LIN {X 0,Y 404.496,Z 624.581,A -85,B 0,C 180,E1 -11091.801,E2 -11091.801} C_VEL
LIN {X 0,Y 405.836,Z 611.424,A -85,B 0,C 180,E1 -11092.797,E2 -11092.797} C_VEL
LIN {X 0,Y 407.026,Z 596.699,A -85,B 0,C 180,E1 -11093.683,E2 -11093.683} C_VEL
LIN {X 0,Y 408.001,Z 581.797,A -85,B 0,C 180,E1 -11094.357,E2 -11094.357} C_VEL
LIN {X 0,Y 408.768,Z 566.165,A -85,B 0,C 180,E1 -11094.844,E2 -11094.844} C_VEL
LIN {X 0,Y 409.775,Z 521.843,A -85,B 0,C 180,E1 -11095.662,E2 -11095.662} C_VEL
LIN {X 0,Y 411.509,Z 429.898,A -85,B 0,C 180,E1 -11097.306,E2 -11097.306} C_VEL
LIN {X 0,Y 405.614,Z 399.49,A -85,B 0,C 180,E1 -11098.332,E2 -11098.332} C_VEL
LIN {X 0,Y 405.096,Z 396.543,A -85,B 0,C 180,E1 -11098.473,E2 -11098.473} C_VEL
LIN {X 0,Y 405.534,Z 388.379,A -85,B 0,C 180,E1 -11099.611,E2 -11099.611} C_VEL
LIN {X 0,Y 402.994,Z 376.938,A -85,B 0,C 180,E1 -11101.546,E2 -11101.546} C_VEL
LIN {X 0,Y 398.838,Z 361.587,A -85,B 0,C 180,E1 -11104.324,E2 -11104.324} C_VEL
LIN {X 0,Y 397.121,Z 355.796,A -85,B 0,C 180,E1 -11105.447,E2 -11105.447} C_VEL
LIN {X 0,Y 397.087,Z 355.636,A -85,B 0,C 180,E1 -11108.853,E2 -11108.853} C_VEL
LIN {X 0,Y 397.053,Z 355.648,A -85,B 0,C 180,E1 -11112.269,E2 -11112.269} C_VEL
LIN {X 0,Y 397.084,Z 355.643,A -85,B 0,C 180,E1 -11115.069,E2 -11115.069} C_VEL
LIN {X 0,Y 397.051,Z 355.65,A -85,B 0,C 180,E1 -11118.024,E2 -11118.024} C_VEL
LIN {X 0,Y 397.089,Z 355.644,A -85,B 0,C 180,E1 -11121.723,E2 -11121.723} C_VEL
LIN {X 0,Y 397.119,Z 355.639,A -85,B 0,C 180,E1 -11125.506,E2 -11125.506} C_VEL
LIN {X 0,Y 397.077,Z 355.639,A -85,B 0,C 180,E1 -11129.117,E2 -11129.117} C_VEL
LIN {X 0,Y 397.099,Z 355.633,A -85,B 0,C 180,E1 -11132.603,E2 -11132.603} C_VEL
LIN {X 0,Y 397.112,Z 355.641,A -85,B 0,C 180,E1 -11135.98,E2 -11135.98} C_VEL
LIN {X 0,Y 397.139,Z 355.64,A -85,B 0,C 180,E1 -11139.705,E2 -11139.705} C_VEL
LIN {X 0,Y 397.182,Z 355.622,A -85,B 0,C 180,E1 -11142.845,E2 -11142.845} C_VEL
LIN {X 0,Y 397.229,Z 355.627,A -85,B 0,C 180,E1 -11146.703,E2 -11146.703} C_VEL
LIN {X 0,Y 397.216,Z 355.619,A -85,B 0,C 180,E1 -11149.809,E2 -11149.809} C_VEL
LIN {X 0,Y 397.335,Z 355.615,A -85,B 0,C 180,E1 -11152.888,E2 -11152.888} C_VEL
LIN {X 0,Y 397.248,Z 355.611,A -85,B 0,C 180,E1 -11154.925,E2 -11154.925} C_VEL
LIN {X 0,Y 397.446,Z 355.602,A -85,B 0,C 180,E1 -11157.973,E2 -11157.973} C_VEL
LIN {X 0,Y 397.577,Z 355.577,A -85,B 0,C 180,E1 -11160,E2 -11160} C_VEL
LIN {X 0,Y 397.37,Z 355.602,A -85,B 0,C 180,E1 -11163.041,E2 -11163.041} C_VEL
LIN {X 0,Y 397.346,Z 355.607,A -85,B 0,C 180,E1 -11166.092,E2 -11166.092} C_VEL
LIN {X 0,Y 397.236,Z 355.617,A -85,B 0,C 180,E1 -11169.162,E2 -11169.162} C_VEL
LIN {X 0,Y 397.22,Z 355.622,A -85,B 0,C 180,E1 -11172.258,E2 -11172.258} C_VEL
LIN {X 0,Y 397.179,Z 355.629,A -85,B 0,C 180,E1 -11175.392,E2 -11175.392} C_VEL
LIN {X 0,Y 397.158,Z 355.631,A -85,B 0,C 180,E1 -11178.574,E2 -11178.574} C_VEL
LIN {X 0,Y 397.109,Z 355.644,A -85,B 0,C 180,E1 -11181.818,E2 -11181.818} C_VEL
LIN {X 0,Y 397.152,Z 355.629,A -85,B 0,C 180,E1 -11185.512,E2 -11185.512} C_VEL
LIN {X 0,Y 397.123,Z 355.642,A -85,B 0,C 180,E1 -11188.543,E2 -11188.543} C_VEL
LIN {X 0,Y 397.078,Z 355.647,A -85,B 0,C 180,E1 -11192.071,E2 -11192.071} C_VEL
LIN {X 0,Y 397.119,Z 355.642,A -85,B 0,C 180,E1 -11195.503,E2 -11195.503} C_VEL
LIN {X 0,Y 397.126,Z 355.616,A -85,B 0,C 180,E1 -11198.861,E2 -11198.861} C_VEL
LIN {X 0,Y 397.071,Z 355.64,A -85,B 0,C 180,E1 -11202.267,E2 -11202.267} C_VEL
LIN {X 0,Y 397.088,Z 355.635,A -85,B 0,C 180,E1 -11205.068,E2 -11205.068} C_VEL
LIN {X 0,Y 397.065,Z 355.633,A -85,B 0,C 180,E1 -11208.021,E2 -11208.021} C_VEL
LIN {X 0,Y 397.131,Z 355.645,A -85,B 0,C 180,E1 -11211.138,E2 -11211.138} C_VEL
LIN {X 0,Y 397.154,Z 355.714,A -85,B 0,C 180,E1 -11215.124,E2 -11215.124} C_VEL
LIN {X 0,Y 397.314,Z 356.566,A -85,B 0,C 180,E1 -11215.372,E2 -11215.372} C_VEL
LIN {X 0,Y 401.916,Z 373.552,A -85,B 0,C 180,E1 -11218.529,E2 -11218.529} C_VEL
LIN {X 0,Y 405.39,Z 387.316,A -85,B 0,C 180,E1 -11220.96,E2 -11220.96} C_VEL
LIN {X 0,Y 405.046,Z 393.159,A -85,B 0,C 180,E1 -11221.805,E2 -11221.805} C_VEL
LIN {X 0,Y 410.902,Z 428.294,A -85,B 0,C 180,E1 -11222.931,E2 -11222.931} C_VEL
LIN {X 0,Y 408.199,Z 565.443,A -85,B 0,C 180,E1 -11225.39,E2 -11225.39} C_VEL
LIN {X 0,Y 407.442,Z 581.285,A -85,B 0,C 180,E1 -11225.88,E2 -11225.88} C_VEL
LIN {X 0,Y 406.442,Z 596.437,A -85,B 0,C 180,E1 -11226.565,E2 -11226.565} C_VEL
LIN {X 0,Y 405.3,Z 610.9,A -85,B 0,C 180,E1 -11227.44,E2 -11227.44} C_VEL
LIN {X 0,Y 403.993,Z 624.081,A -85,B 0,C 180,E1 -11228.439,E2 -11228.439} C_VEL
LIN {X 0,Y 402.589,Z 637.469,A -85,B 0,C 180,E1 -11229.699,E2 -11229.699} C_VEL
LIN {X 0,Y 401.232,Z 649.387,A -85,B 0,C 180,E1 -11231.061,E2 -11231.061} C_VEL
LIN {X 0,Y 399.9,Z 660.685,A -85,B 0,C 180,E1 -11232.617,E2 -11232.617} C_VEL
LIN {X 0,Y 398.64,Z 671.405,A -85,B 0,C 180,E1 -11234.404,E2 -11234.404} C_VEL
LIN {X 0,Y 397.674,Z 680.308,A -85,B 0,C 180,E1 -11236.198,E2 -11236.198} C_VEL
LIN {X 0,Y 396.924,Z 688.618,A -85,B 0,C 180,E1 -11238.251,E2 -11238.251} C_VEL
LIN {X 0,Y 396.32,Z 695.281,A -85,B 0,C 180,E1 -11240.302,E2 -11240.302} C_VEL
LIN {X 0,Y 396.016,Z 700.482,A -85,B 0,C 180,E1 -11242.351,E2 -11242.351} C_VEL
LIN {X 0,Y 395.859,Z 703.468,A -85,B 0,C 180,E1 -11243.885,E2 -11243.885} C_VEL
LIN {X 0,Y 395.745,Z 706.394,A -85,B 0,C 180,E1 -11245.927,E2 -11245.927} C_VEL
LIN {X 0,Y 395.77,Z 708.14,A -85,B 0,C 180,E1 -11247.965,E2 -11247.965} C_VEL
LIN {X 0,Y 395.723,Z 708.736,A -85,B 0,C 180,E1 -11250,E2 -11250} C_VEL
LIN {X 0,Y 395.772,Z 708.14,A -85,B 0,C 180,E1 -11252.035,E2 -11252.035} C_VEL
LIN {X 0,Y 395.745,Z 706.393,A -85,B 0,C 180,E1 -11254.074,E2 -11254.074} C_VEL
LIN {X 0,Y 395.858,Z 703.37,A -85,B 0,C 180,E1 -11256.167,E2 -11256.167} C_VEL
LIN {X 0,Y 396.074,Z 699.273,A -85,B 0,C 180,E1 -11258.161,E2 -11258.161} C_VEL
LIN {X 0,Y 396.424,Z 693.73,A -85,B 0,C 180,E1 -11260.212,E2 -11260.212} C_VEL
LIN {X 0,Y 397.131,Z 686.671,A -85,B 0,C 180,E1 -11262.261,E2 -11262.261} C_VEL
LIN {X 0,Y 397.811,Z 679.217,A -85,B 0,C 180,E1 -11264.033,E2 -11264.033} C_VEL
LIN {X 0,Y 398.82,Z 669.954,A -85,B 0,C 180,E1 -11265.851,E2 -11265.851} C_VEL
LIN {X 0,Y 399.876,Z 660.639,A -85,B 0,C 180,E1 -11267.385,E2 -11267.385} C_VEL
LIN {X 0,Y 401.249,Z 649.268,A -85,B 0,C 180,E1 -11268.946,E2 -11268.946} C_VEL
LIN {X 0,Y 402.557,Z 637.39,A -85,B 0,C 180,E1 -11270.303,E2 -11270.303} C_VEL
LIN {X 0,Y 404.026,Z 623.994,A -85,B 0,C 180,E1 -11271.56,E2 -11271.56} C_VEL
LIN {X 0,Y 405.321,Z 610.799,A -85,B 0,C 180,E1 -11272.559,E2 -11272.559} C_VEL
LIN {X 0,Y 406.496,Z 596.286,A -85,B 0,C 180,E1 -11273.432,E2 -11273.432} C_VEL
LIN {X 0,Y 407.456,Z 581.386,A -85,B 0,C 180,E1 -11274.106,E2 -11274.106} C_VEL
LIN {X 0,Y 408.166,Z 566.338,A -85,B 0,C 180,E1 -11274.578,E2 -11274.578} C_VEL
LIN {X 0,Y 409.234,Z 520.04,A -85,B 0,C 180,E1 -11275.46,E2 -11275.46} C_VEL
LIN {X 0,Y 413.083,Z 440.948,A -85,B 0,C 180,E1 -11277.431,E2 -11277.431} C_VEL
LIN {X 0,Y 413.644,Z 427.571,A -85,B 0,C 180,E1 -11277.796,E2 -11277.796} C_VEL
LIN {X 0,Y 411.809,Z 413.574,A -85,B 0,C 180,E1 -11278.454,E2 -11278.454} C_VEL
LIN {X 0,Y 409.144,Z 400.165,A -85,B 0,C 180,E1 -11279.23,E2 -11279.23} C_VEL
LIN {X 0,Y 408.97,Z 398.32,A -85,B 0,C 180,E1 -11279.396,E2 -11279.396} C_VEL
LIN {X 0,Y 409.415,Z 395.73,A -85,B 0,C 180,E1 -11279.856,E2 -11279.856} C_VEL
LIN {X 0,Y 408.208,Z 388.55,A -85,B 0,C 180,E1 -11281.555,E2 -11281.555} C_VEL
LIN {X 0,Y 406.088,Z 380.467,A -85,B 0,C 180,E1 -11283.828,E2 -11283.828} C_VEL
LIN {X 0,Y 404.473,Z 375.21,A -85,B 0,C 180,E1 -11285.597,E2 -11285.597} C_VEL
LIN {X 0,Y 402.791,Z 370.256,A -85,B 0,C 180,E1 -11287.64,E2 -11287.64} C_VEL
LIN {X 0,Y 401.442,Z 366.5,A -85,B 0,C 180,E1 -11289.619,E2 -11289.619} C_VEL
LIN {X 0,Y 400.118,Z 362.916,A -85,B 0,C 180,E1 -11292.462,E2 -11292.462} C_VEL
LIN {X 0,Y 399.433,Z 361.71,A -85,B 0,C 180,E1 -11294.733,E2 -11294.733} C_VEL
LIN {X 0,Y 399.379,Z 361.646,A -85,B 0,C 180,E1 -11296.663,E2 -11296.663} C_VEL
LIN {X 0,Y 399.947,Z 362.755,A -85,B 0,C 180,E1 -11299.079,E2 -11299.079} C_VEL
LIN {X 0,Y 400.562,Z 364.58,A -85,B 0,C 180,E1 -11300.829,E2 -11300.829} C_VEL
LIN {X 0,Y 401.718,Z 367.697,A -85,B 0,C 180,E1 -11302.955,E2 -11302.955} C_VEL
LIN {X 0,Y 403.088,Z 371.791,A -85,B 0,C 180,E1 -11305.031,E2 -11305.031} C_VEL
LIN {X 0,Y 404.542,Z 376.587,A -85,B 0,C 180,E1 -11306.986,E2 -11306.986} C_VEL
LIN {X 0,Y 406.267,Z 383.464,A -85,B 0,C 180,E1 -11309.316,E2 -11309.316} C_VEL
LIN {X 0,Y 407.786,Z 391.148,A -85,B 0,C 180,E1 -11311.518,E2 -11311.518} C_VEL
LIN {X 0,Y 407.932,Z 394.194,A -85,B 0,C 180,E1 -11312.279,E2 -11312.279} C_VEL
LIN {X 0,Y 407.212,Z 399.018,A -85,B 0,C 180,E1 -11313.234,E2 -11313.234} C_VEL
LIN {X 0,Y 410.848,Z 414.131,A -85,B 0,C 180,E1 -11314.275,E2 -11314.275} C_VEL
LIN {X 0,Y 413.382,Z 428.709,A -85,B 0,C 180,E1 -11315.09,E2 -11315.09} C_VEL
LIN {X 0,Y 408.751,Z 507.668,A -85,B 0,C 180,E1 -11317.274,E2 -11317.274} C_VEL
LIN {X 0,Y 406.938,Z 545.844,A -85,B 0,C 180,E1 -11318.337,E2 -11318.337} C_VEL
LIN {X 0,Y 405.969,Z 560.659,A -85,B 0,C 180,E1 -11318.948,E2 -11318.948} C_VEL
LIN {X 0,Y 405.03,Z 573.977,A -85,B 0,C 180,E1 -11319.694,E2 -11319.694} C_VEL
LIN {X 0,Y 403.786,Z 588.032,A -85,B 0,C 180,E1 -11320.689,E2 -11320.689} C_VEL
LIN {X 0,Y 402.511,Z 600.735,A -85,B 0,C 180,E1 -11321.814,E2 -11321.814} C_VEL
LIN {X 0,Y 401.412,Z 612.369,A -85,B 0,C 180,E1 -11323.078,E2 -11323.078} C_VEL
LIN {X 0,Y 400.281,Z 623.016,A -85,B 0,C 180,E1 -11324.469,E2 -11324.469} C_VEL
LIN {X 0,Y 399.173,Z 632.705,A -85,B 0,C 180,E1 -11325.99,E2 -11325.99} C_VEL
LIN {X 0,Y 398.156,Z 641.988,A -85,B 0,C 180,E1 -11327.771,E2 -11327.771} C_VEL
LIN {X 0,Y 397.5,Z 648.472,A -85,B 0,C 180,E1 -11329.301,E2 -11329.301} C_VEL
LIN {X 0,Y 397.002,Z 653.817,A -85,B 0,C 180,E1 -11330.832,E2 -11330.832} C_VEL
LIN {X 0,Y 396.499,Z 659.433,A -85,B 0,C 180,E1 -11332.873,E2 -11332.873} C_VEL
LIN {X 0,Y 396.354,Z 661.618,A -85,B 0,C 180,E1 -11333.893,E2 -11333.893} C_VEL
LIN {X 0,Y 396.1,Z 663.414,A -85,B 0,C 180,E1 -11334.91,E2 -11334.91} C_VEL
LIN {X 0,Y 396.128,Z 664.813,A -85,B 0,C 180,E1 -11335.931,E2 -11335.931} C_VEL
LIN {X 0,Y 395.943,Z 666.546,A -85,B 0,C 180,E1 -11337.966,E2 -11337.966} C_VEL
LIN {X 0,Y 395.828,Z 666.851,A -85,B 0,C 180,E1 -11340,E2 -11340} C_VEL
LIN {X 0,Y 395.921,Z 665.725,A -85,B 0,C 180,E1 -11342.035,E2 -11342.035} C_VEL
LIN {X 0,Y 395.951,Z 664.627,A -85,B 0,C 180,E1 -11343.053,E2 -11343.053} C_VEL
LIN {X 0,Y 396.06,Z 661.325,A -85,B 0,C 180,E1 -11345.09,E2 -11345.09} C_VEL
LIN {X 0,Y 396.294,Z 656.472,A -85,B 0,C 180,E1 -11347.131,E2 -11347.131} C_VEL
LIN {X 0,Y 396.497,Z 651.676,A -85,B 0,C 180,E1 -11348.666,E2 -11348.666} C_VEL
LIN {X 0,Y 396.995,Z 644.761,A -85,B 0,C 180,E1 -11350.455,E2 -11350.455} C_VEL
LIN {X 0,Y 397.633,Z 636.163,A -85,B 0,C 180,E1 -11352.245,E2 -11352.245} C_VEL
LIN {X 0,Y 398.303,Z 627.118,A -85,B 0,C 180,E1 -11353.787,E2 -11353.787} C_VEL
LIN {X 0,Y 399.109,Z 616.263,A -85,B 0,C 180,E1 -11355.316,E2 -11355.316} C_VEL
LIN {X 0,Y 400.065,Z 604.127,A -85,B 0,C 180,E1 -11356.718,E2 -11356.718} C_VEL
LIN {X 0,Y 401.011,Z 592.05,A -85,B 0,C 180,E1 -11357.861,E2 -11357.861} C_VEL
LIN {X 0,Y 401.9,Z 578.996,A -85,B 0,C 180,E1 -11358.866,E2 -11358.866} C_VEL
LIN {X 0,Y 402.718,Z 565.293,A -85,B 0,C 180,E1 -11359.696,E2 -11359.696} C_VEL
LIN {X 0,Y 403.402,Z 550.716,A -85,B 0,C 180,E1 -11360.359,E2 -11360.359} C_VEL
LIN {X 0,Y 403.957,Z 535.718,A -85,B 0,C 180,E1 -11360.828,E2 -11360.828} C_VEL
LIN {X 0,Y 406.903,Z 425.509,A -85,B 0,C 180,E1 -11363.296,E2 -11363.296} C_VEL
LIN {X 0,Y 402.07,Z 397.746,A -85,B 0,C 180,E1 -11364.253,E2 -11364.253} C_VEL
LIN {X 0,Y 403.355,Z 382.587,A -85,B 0,C 180,E1 -11366.938,E2 -11366.938} C_VEL
LIN {X 0,Y 400.277,Z 368.92,A -85,B 0,C 180,E1 -11369.703,E2 -11369.703} C_VEL
LIN {X 0,Y 397.147,Z 356.013,A -85,B 0,C 180,E1 -11372.44,E2 -11372.44} C_VEL
LIN {X 0,Y 397.114,Z 355.658,A -85,B 0,C 180,E1 -11372.669,E2 -11372.669} C_VEL
LIN {X 0,Y 397.092,Z 355.648,A -85,B 0,C 180,E1 -11375.736,E2 -11375.736} C_VEL
LIN {X 0,Y 397.091,Z 355.646,A -85,B 0,C 180,E1 -11378.854,E2 -11378.854} C_VEL
LIN {X 0,Y 397.053,Z 355.634,A -85,B 0,C 180,E1 -11382.269,E2 -11382.269} C_VEL
LIN {X 0,Y 397.084,Z 355.648,A -85,B 0,C 180,E1 -11385.069,E2 -11385.069} C_VEL
LIN {X 0,Y 397.051,Z 355.645,A -85,B 0,C 180,E1 -11388.024,E2 -11388.024} C_VEL
LIN {X 0,Y 397.088,Z 355.64,A -85,B 0,C 180,E1 -11391.146,E2 -11391.146} C_VEL
LIN {X 0,Y 397.142,Z 355.808,A -85,B 0,C 180,E1 -11394.665,E2 -11394.665} C_VEL
LIN {X 0,Y 401.061,Z 369.651,A -85,B 0,C 180,E1 -11397.26,E2 -11397.26} C_VEL
LIN {X 0,Y 405.209,Z 386.155,A -85,B 0,C 180,E1 -11400.136,E2 -11400.136} C_VEL
LIN {X 0,Y 405.518,Z 388.974,A -85,B 0,C 180,E1 -11400.579,E2 -11400.579} C_VEL
LIN {X 0,Y 405.126,Z 396.894,A -85,B 0,C 180,E1 -11401.665,E2 -11401.665} C_VEL
LIN {X 0,Y 411.471,Z 429.941,A -85,B 0,C 180,E1 -11402.791,E2 -11402.791} C_VEL
LIN {X 0,Y 409.495,Z 534.502,A -85,B 0,C 180,E1 -11404.66,E2 -11404.66} C_VEL
LIN {X 0,Y 408.796,Z 566.283,A -85,B 0,C 180,E1 -11405.259,E2 -11405.259} C_VEL
LIN {X 0,Y 408.024,Z 581.59,A -85,B 0,C 180,E1 -11405.735,E2 -11405.735} C_VEL
LIN {X 0,Y 407.742,Z 585.778,A -85,B 0,C 180,E1 -11405.903,E2 -11405.903} C_VEL
LIN {X 0,Y 406.861,Z 591.448,A -85,B 0,C 180,E1 -11406.121,E2 -11406.121} C_VEL
LIN {X 0,Y 403.635,Z 600.495,A -85,B 0,C 180,E1 -11406.435,E2 -11406.435} C_VEL
LIN {X 0,Y 400.137,Z 609.404,A -85,B 0,C 180,E1 -11406.813,E2 -11406.813} C_VEL
LIN {X 0,Y 398.893,Z 614.699,A -85,B 0,C 180,E1 -11407.141,E2 -11407.141} C_VEL
LIN {X 0,Y 397.495,Z 627.829,A -85,B 0,C 180,E1 -11408.204,E2 -11408.204} C_VEL
LIN {X 0,Y 396.009,Z 640.681,A -85,B 0,C 180,E1 -11409.482,E2 -11409.482} C_VEL
LIN {X 0,Y 394.566,Z 652.345,A -85,B 0,C 180,E1 -11410.881,E2 -11410.881} C_VEL
LIN {X 0,Y 393.264,Z 662.425,A -85,B 0,C 180,E1 -11412.313,E2 -11412.313} C_VEL
LIN {X 0,Y 391.942,Z 673.038,A -85,B 0,C 180,E1 -11414.13,E2 -11414.13} C_VEL
LIN {X 0,Y 390.839,Z 682.096,A -85,B 0,C 180,E1 -11416.004,E2 -11416.004} C_VEL
LIN {X 0,Y 390.028,Z 690.139,A -85,B 0,C 180,E1 -11418.04,E2 -11418.04} C_VEL
LIN {X 0,Y 389.319,Z 696.765,A -85,B 0,C 180,E1 -11420.125,E2 -11420.125} C_VEL
LIN {X 0,Y 388.953,Z 701.954,A -85,B 0,C 180,E1 -11422.211,E2 -11422.211} C_VEL
LIN {X 0,Y 388.75,Z 705.136,A -85,B 0,C 180,E1 -11423.889,E2 -11423.889} C_VEL
LIN {X 0,Y 388.665,Z 707.876,A -85,B 0,C 180,E1 -11425.852,E2 -11425.852} C_VEL
LIN {X 0,Y 388.613,Z 709.638,A -85,B 0,C 180,E1 -11427.927,E2 -11427.927} C_VEL
LIN {X 0,Y 388.639,Z 710.248,A -85,B 0,C 180,E1 -11430,E2 -11430} C_VEL
LIN {X 0,Y 388.613,Z 709.679,A -85,B 0,C 180,E1 -11432.073,E2 -11432.073} C_VEL
LIN {X 0,Y 388.667,Z 707.974,A -85,B 0,C 180,E1 -11434.148,E2 -11434.148} C_VEL
LIN {X 0,Y 388.797,Z 705.1,A -85,B 0,C 180,E1 -11436.226,E2 -11436.226} C_VEL
LIN {X 0,Y 389.029,Z 700.989,A -85,B 0,C 180,E1 -11438.31,E2 -11438.31} C_VEL
LIN {X 0,Y 389.413,Z 695.53,A -85,B 0,C 180,E1 -11440.397,E2 -11440.397} C_VEL
LIN {X 0,Y 390.186,Z 688.578,A -85,B 0,C 180,E1 -11442.482,E2 -11442.482} C_VEL
LIN {X 0,Y 390.955,Z 681.137,A -85,B 0,C 180,E1 -11444.31,E2 -11444.31} C_VEL
LIN {X 0,Y 392.046,Z 672.172,A -85,B 0,C 180,E1 -11446.132,E2 -11446.132} C_VEL
LIN {X 0,Y 393.461,Z 661.337,A -85,B 0,C 180,E1 -11447.946,E2 -11447.946} C_VEL
LIN {X 0,Y 394.842,Z 650.083,A -85,B 0,C 180,E1 -11449.513,E2 -11449.513} C_VEL
LIN {X 0,Y 396.338,Z 638.01,A -85,B 0,C 180,E1 -11450.908,E2 -11450.908} C_VEL
LIN {X 0,Y 397.896,Z 624.545,A -85,B 0,C 180,E1 -11452.182,E2 -11452.182} C_VEL
LIN {X 0,Y 399.282,Z 611.381,A -85,B 0,C 180,E1 -11453.193,E2 -11453.193} C_VEL
LIN {X 0,Y 400.453,Z 597.652,A -85,B 0,C 180,E1 -11454.039,E2 -11454.039} C_VEL
LIN {X 0,Y 401.511,Z 582.43,A -85,B 0,C 180,E1 -11454.749,E2 -11454.749} C_VEL
LIN {X 0,Y 402.299,Z 567.399,A -85,B 0,C 180,E1 -11455.237,E2 -11455.237} C_VEL
LIN {X 0,Y 402.986,Z 539.519,A -85,B 0,C 180,E1 -11455.779,E2 -11455.779} C_VEL
LIN {X 0,Y 405.202,Z 431.044,A -85,B 0,C 180,E1 -11457.742,E2 -11457.742} C_VEL
LIN {X 0,Y 399.57,Z 401.702,A -85,B 0,C 180,E1 -11458.753,E2 -11458.753} C_VEL
LIN {X 0,Y 398.562,Z 396.728,A -85,B 0,C 180,E1 -11458.956,E2 -11458.956} C_VEL
LIN {X 0,Y 398.859,Z 389.896,A -85,B 0,C 180,E1 -11459.911,E2 -11459.911} C_VEL
LIN {X 0,Y 395.09,Z 374.079,A -85,B 0,C 180,E1 -11462.653,E2 -11462.653} C_VEL
LIN {X 0,Y 391.427,Z 361.156,A -85,B 0,C 180,E1 -11465.068,E2 -11465.068} C_VEL
LIN {X 0,Y 390.058,Z 356.681,A -85,B 0,C 180,E1 -11465.967,E2 -11465.967} C_VEL
LIN {X 0,Y 390.032,Z 356.511,A -85,B 0,C 180,E1 -11469.211,E2 -11469.211} C_VEL
LIN {X 0,Y 390.029,Z 356.523,A -85,B 0,C 180,E1 -11472.372,E2 -11472.372} C_VEL
LIN {X 0,Y 390.041,Z 356.521,A -85,B 0,C 180,E1 -11475.354,E2 -11475.354} C_VEL
LIN {X 0,Y 390.014,Z 356.526,A -85,B 0,C 180,E1 -11478.184,E2 -11478.184} C_VEL
LIN {X 0,Y 390.056,Z 356.516,A -85,B 0,C 180,E1 -11480.903,E2 -11480.903} C_VEL
LIN {X 0,Y 390.07,Z 356.512,A -85,B 0,C 180,E1 -11484.791,E2 -11484.791} C_VEL
LIN {X 0,Y 390.022,Z 356.516,A -85,B 0,C 180,E1 -11488.495,E2 -11488.495} C_VEL
LIN {X 0,Y 390.037,Z 356.515,A -85,B 0,C 180,E1 -11492.064,E2 -11492.064} C_VEL
LIN {X 0,Y 390.044,Z 356.527,A -85,B 0,C 180,E1 -11495.517,E2 -11495.517} C_VEL
LIN {X 0,Y 390.056,Z 356.514,A -85,B 0,C 180,E1 -11498.878,E2 -11498.878} C_VEL
LIN {X 0,Y 390.112,Z 356.505,A -85,B 0,C 180,E1 -11502.166,E2 -11502.166} C_VEL
LIN {X 0,Y 390.145,Z 356.51,A -85,B 0,C 180,E1 -11505.393,E2 -11505.393} C_VEL
LIN {X 0,Y 390.147,Z 356.497,A -85,B 0,C 180,E1 -11508.571,E2 -11508.571} C_VEL
LIN {X 0,Y 390.271,Z 356.495,A -85,B 0,C 180,E1 -11512.071,E2 -11512.071} C_VEL
LIN {X 0,Y 390.221,Z 356.486,A -85,B 0,C 180,E1 -11514.833,E2 -11514.833} C_VEL
LIN {X 0,Y 390.413,Z 356.478,A -85,B 0,C 180,E1 -11517.937,E2 -11517.937} C_VEL
LIN {X 0,Y 390.547,Z 356.452,A -85,B 0,C 180,E1 -11520,E2 -11520} C_VEL
LIN {X 0,Y 390.304,Z 356.483,A -85,B 0,C 180,E1 -11523.096,E2 -11523.096} C_VEL
LIN {X 0,Y 390.3,Z 356.484,A -85,B 0,C 180,E1 -11526.202,E2 -11526.202} C_VEL
LIN {X 0,Y 390.194,Z 356.496,A -85,B 0,C 180,E1 -11529.329,E2 -11529.329} C_VEL
LIN {X 0,Y 390.171,Z 356.501,A -85,B 0,C 180,E1 -11532.483,E2 -11532.483} C_VEL
LIN {X 0,Y 390.14,Z 356.51,A -85,B 0,C 180,E1 -11535.677,E2 -11535.677} C_VEL
LIN {X 0,Y 390.103,Z 356.505,A -85,B 0,C 180,E1 -11538.922,E2 -11538.922} C_VEL
LIN {X 0,Y 390.047,Z 356.522,A -85,B 0,C 180,E1 -11542.234,E2 -11542.234} C_VEL
LIN {X 0,Y 390.119,Z 356.507,A -85,B 0,C 180,E1 -11545.743,E2 -11545.743} C_VEL
LIN {X 0,Y 390.059,Z 356.514,A -85,B 0,C 180,E1 -11549.109,E2 -11549.109} C_VEL
LIN {X 0,Y 390.043,Z 356.527,A -85,B 0,C 180,E1 -11552.721,E2 -11552.721} C_VEL
LIN {X 0,Y 390.056,Z 356.522,A -85,B 0,C 180,E1 -11555.825,E2 -11555.825} C_VEL
LIN {X 0,Y 390.066,Z 356.489,A -85,B 0,C 180,E1 -11559.218,E2 -11559.218} C_VEL
LIN {X 0,Y 390.044,Z 356.516,A -85,B 0,C 180,E1 -11562.374,E2 -11562.374} C_VEL
LIN {X 0,Y 390.045,Z 356.509,A -85,B 0,C 180,E1 -11565.355,E2 -11565.355} C_VEL
LIN {X 0,Y 390.03,Z 356.512,A -85,B 0,C 180,E1 -11568.187,E2 -11568.187} C_VEL
LIN {X 0,Y 390.09,Z 356.521,A -85,B 0,C 180,E1 -11570.908,E2 -11570.908} C_VEL
LIN {X 0,Y 390.137,Z 356.736,A -85,B 0,C 180,E1 -11574.799,E2 -11574.799} C_VEL
LIN {X 0,Y 394.94,Z 374.772,A -85,B 0,C 180,E1 -11578.24,E2 -11578.24} C_VEL
LIN {X 0,Y 398.368,Z 388.354,A -85,B 0,C 180,E1 -11580.688,E2 -11580.688} C_VEL
LIN {X 0,Y 398.427,Z 391.59,A -85,B 0,C 180,E1 -11581.199,E2 -11581.199} C_VEL
LIN {X 0,Y 398.563,Z 393.322,A -85,B 0,C 180,E1 -11581.314,E2 -11581.314} C_VEL
LIN {X 0,Y 404.49,Z 428.328,A -85,B 0,C 180,E1 -11582.464,E2 -11582.464} C_VEL
LIN {X 0,Y 402.199,Z 547.523,A -85,B 0,C 180,E1 -11584.618,E2 -11584.618} C_VEL
LIN {X 0,Y 401.674,Z 567.848,A -85,B 0,C 180,E1 -11585.032,E2 -11585.032} C_VEL
LIN {X 0,Y 400.883,Z 583.023,A -85,B 0,C 180,E1 -11585.536,E2 -11585.536} C_VEL
LIN {X 0,Y 399.871,Z 597.345,A -85,B 0,C 180,E1 -11586.209,E2 -11586.209} C_VEL
LIN {X 0,Y 398.757,Z 610.94,A -85,B 0,C 180,E1 -11587.049,E2 -11587.049} C_VEL
LIN {X 0,Y 397.36,Z 624.115,A -85,B 0,C 180,E1 -11588.06,E2 -11588.06} C_VEL
LIN {X 0,Y 395.907,Z 637.497,A -85,B 0,C 180,E1 -11589.341,E2 -11589.341} C_VEL
LIN {X 0,Y 394.533,Z 649.108,A -85,B 0,C 180,E1 -11590.686,E2 -11590.686} C_VEL
LIN {X 0,Y 393.084,Z 660.707,A -85,B 0,C 180,E1 -11592.305,E2 -11592.305} C_VEL
LIN {X 0,Y 391.737,Z 671.425,A -85,B 0,C 180,E1 -11594.122,E2 -11594.122} C_VEL
LIN {X 0,Y 390.708,Z 680.547,A -85,B 0,C 180,E1 -11595.999,E2 -11595.999} C_VEL
LIN {X 0,Y 389.92,Z 688.635,A -85,B 0,C 180,E1 -11598.037,E2 -11598.037} C_VEL
LIN {X 0,Y 389.273,Z 695.297,A -85,B 0,C 180,E1 -11600.124,E2 -11600.124} C_VEL
LIN {X 0,Y 388.948,Z 700.497,A -85,B 0,C 180,E1 -11602.211,E2 -11602.211} C_VEL
LIN {X 0,Y 388.772,Z 703.624,A -85,B 0,C 180,E1 -11603.856,E2 -11603.856} C_VEL
LIN {X 0,Y 388.67,Z 706.408,A -85,B 0,C 180,E1 -11605.852,E2 -11605.852} C_VEL
LIN {X 0,Y 388.666,Z 708.154,A -85,B 0,C 180,E1 -11607.928,E2 -11607.928} C_VEL
LIN {X 0,Y 388.638,Z 708.75,A -85,B 0,C 180,E1 -11610,E2 -11610} C_VEL
LIN {X 0,Y 388.668,Z 708.153,A -85,B 0,C 180,E1 -11612.073,E2 -11612.073} C_VEL
LIN {X 0,Y 388.67,Z 706.406,A -85,B 0,C 180,E1 -11614.148,E2 -11614.148} C_VEL
LIN {X 0,Y 388.775,Z 703.473,A -85,B 0,C 180,E1 -11616.227,E2 -11616.227} C_VEL
LIN {X 0,Y 389.021,Z 699.287,A -85,B 0,C 180,E1 -11618.31,E2 -11618.31} C_VEL
LIN {X 0,Y 389.378,Z 693.744,A -85,B 0,C 180,E1 -11620.399,E2 -11620.399} C_VEL
LIN {X 0,Y 390.107,Z 686.687,A -85,B 0,C 180,E1 -11622.485,E2 -11622.485} C_VEL
LIN {X 0,Y 390.866,Z 679.233,A -85,B 0,C 180,E1 -11624.287,E2 -11624.287} C_VEL
LIN {X 0,Y 391.946,Z 669.971,A -85,B 0,C 180,E1 -11626.137,E2 -11626.137} C_VEL
LIN {X 0,Y 393.064,Z 660.657,A -85,B 0,C 180,E1 -11627.696,E2 -11627.696} C_VEL
LIN {X 0,Y 394.602,Z 648.646,A -85,B 0,C 180,E1 -11629.362,E2 -11629.362} C_VEL
LIN {X 0,Y 396.05,Z 636.18,A -85,B 0,C 180,E1 -11630.788,E2 -11630.788} C_VEL
LIN {X 0,Y 397.413,Z 624.02,A -85,B 0,C 180,E1 -11631.937,E2 -11631.937} C_VEL
LIN {X 0,Y 398.775,Z 610.829,A -85,B 0,C 180,E1 -11632.95,E2 -11632.95} C_VEL
LIN {X 0,Y 399.991,Z 596.323,A -85,B 0,C 180,E1 -11633.836,E2 -11633.836} C_VEL
LIN {X 0,Y 401.011,Z 580.981,A -85,B 0,C 180,E1 -11634.538,E2 -11634.538} C_VEL
LIN {X 0,Y 401.728,Z 566.41,A -85,B 0,C 180,E1 -11634.999,E2 -11634.999} C_VEL
LIN {X 0,Y 402.643,Z 533.192,A -85,B 0,C 180,E1 -11635.664,E2 -11635.664} C_VEL
LIN {X 0,Y 406.207,Z 461.684,A -85,B 0,C 180,E1 -11637.478,E2 -11637.478} C_VEL
LIN {X 0,Y 408.027,Z 429.238,A -85,B 0,C 180,E1 -11638.352,E2 -11638.352} C_VEL
LIN {X 0,Y 406.223,Z 414.882,A -85,B 0,C 180,E1 -11639.061,E2 -11639.061} C_VEL
LIN {X 0,Y 403.694,Z 401.798,A -85,B 0,C 180,E1 -11639.863,E2 -11639.863} C_VEL
LIN {X 0,Y 403.123,Z 398.596,A -85,B 0,C 180,E1 -11640.118,E2 -11640.118} C_VEL
LIN {X 0,Y 402.505,Z 394.045,A -85,B 0,C 180,E1 -11641.177,E2 -11641.177} C_VEL
LIN {X 0,Y 400.592,Z 385.854,A -85,B 0,C 180,E1 -11643.45,E2 -11643.45} C_VEL
LIN {X 0,Y 398.763,Z 379.527,A -85,B 0,C 180,E1 -11645.564,E2 -11645.564} C_VEL
LIN {X 0,Y 397.156,Z 374.624,A -85,B 0,C 180,E1 -11647.626,E2 -11647.626} C_VEL
LIN {X 0,Y 395.517,Z 370.097,A -85,B 0,C 180,E1 -11650.176,E2 -11650.176} C_VEL
LIN {X 0,Y 394.553,Z 367.263,A -85,B 0,C 180,E1 -11652.6,E2 -11652.6} C_VEL
LIN {X 0,Y 393.979,Z 366.289,A -85,B 0,C 180,E1 -11654.476,E2 -11654.476} C_VEL
LIN {X 0,Y 393.891,Z 366.186,A -85,B 0,C 180,E1 -11657.016,E2 -11657.016} C_VEL
LIN {X 0,Y 394.282,Z 366.953,A -85,B 0,C 180,E1 -11658.737,E2 -11658.737} C_VEL
LIN {X 0,Y 395.248,Z 369.745,A -85,B 0,C 180,E1 -11661.479,E2 -11661.479} C_VEL
LIN {X 0,Y 396.384,Z 372.82,A -85,B 0,C 180,E1 -11663.469,E2 -11663.469} C_VEL
LIN {X 0,Y 398.038,Z 378.346,A -85,B 0,C 180,E1 -11666.085,E2 -11666.085} C_VEL
LIN {X 0,Y 399.887,Z 385.679,A -85,B 0,C 180,E1 -11668.772,E2 -11668.772} C_VEL
LIN {X 0,Y 401.373,Z 393.367,A -85,B 0,C 180,E1 -11671.104,E2 -11671.104} C_VEL
LIN {X 0,Y 401.655,Z 395.99,A -85,B 0,C 180,E1 -11671.808,E2 -11671.808} C_VEL
LIN {X 0,Y 401.271,Z 399.04,A -85,B 0,C 180,E1 -11672.435,E2 -11672.435} C_VEL
LIN {X 0,Y 404.43,Z 411.898,A -85,B 0,C 180,E1 -11673.412,E2 -11673.412} C_VEL
LIN {X 0,Y 407.398,Z 427.651,A -85,B 0,C 180,E1 -11674.383,E2 -11674.383} C_VEL
LIN {X 0,Y 407.701,Z 430.811,A -85,B 0,C 180,E1 -11674.538,E2 -11674.538} C_VEL
LIN {X 0,Y 402.599,Z 510.198,A -85,B 0,C 180,E1 -11676.805,E2 -11676.805} C_VEL
LIN {X 0,Y 400.743,Z 546.291,A -85,B 0,C 180,E1 -11677.849,E2 -11677.849} C_VEL
LIN {X 0,Y 399.712,Z 561.158,A -85,B 0,C 180,E1 -11678.481,E2 -11678.481} C_VEL
LIN {X 0,Y 398.534,Z 576.074,A -85,B 0,C 180,E1 -11679.348,E2 -11679.348} C_VEL
LIN {X 0,Y 397.229,Z 589.675,A -85,B 0,C 180,E1 -11680.357,E2 -11680.357} C_VEL
LIN {X 0,Y 395.789,Z 603.372,A -85,B 0,C 180,E1 -11681.628,E2 -11681.628} C_VEL
LIN {X 0,Y 394.48,Z 615.646,A -85,B 0,C 180,E1 -11683.038,E2 -11683.038} C_VEL
LIN {X 0,Y 393.312,Z 625.791,A -85,B 0,C 180,E1 -11684.453,E2 -11684.453} C_VEL
LIN {X 0,Y 392.161,Z 635.047,A -85,B 0,C 180,E1 -11685.999,E2 -11685.999} C_VEL
LIN {X 0,Y 391.145,Z 643.899,A -85,B 0,C 180,E1 -11687.812,E2 -11687.812} C_VEL
LIN {X 0,Y 390.372,Z 651.054,A -85,B 0,C 180,E1 -11689.628,E2 -11689.628} C_VEL
LIN {X 0,Y 389.852,Z 656.027,A -85,B 0,C 180,E1 -11691.186,E2 -11691.186} C_VEL
LIN {X 0,Y 389.418,Z 660.638,A -85,B 0,C 180,E1 -11693.031,E2 -11693.031} C_VEL
LIN {X 0,Y 389.048,Z 663.922,A -85,B 0,C 180,E1 -11694.818,E2 -11694.818} C_VEL
LIN {X 0,Y 389.009,Z 666.299,A -85,B 0,C 180,E1 -11696.893,E2 -11696.893} C_VEL
LIN {X 0,Y 388.785,Z 667.257,A -85,B 0,C 180,E1 -11698.964,E2 -11698.964} C_VEL
LIN {X 0,Y 388.773,Z 666.779,A -85,B 0,C 180,E1 -11701.036,E2 -11701.036} C_VEL
LIN {X 0,Y 388.854,Z 666.002,A -85,B 0,C 180,E1 -11702.072,E2 -11702.072} C_VEL
LIN {X 0,Y 388.845,Z 663.368,A -85,B 0,C 180,E1 -11704.146,E2 -11704.146} C_VEL
LIN {X 0,Y 389.047,Z 660.381,A -85,B 0,C 180,E1 -11705.702,E2 -11705.702} C_VEL
LIN {X 0,Y 389.232,Z 656.528,A -85,B 0,C 180,E1 -11707.261,E2 -11707.261} C_VEL
LIN {X 0,Y 389.443,Z 651.668,A -85,B 0,C 180,E1 -11708.824,E2 -11708.824} C_VEL
LIN {X 0,Y 389.976,Z 644.653,A -85,B 0,C 180,E1 -11710.645,E2 -11710.645} C_VEL
LIN {X 0,Y 390.514,Z 637.27,A -85,B 0,C 180,E1 -11712.208,E2 -11712.208} C_VEL
LIN {X 0,Y 391.301,Z 627.448,A -85,B 0,C 180,E1 -11713.927,E2 -11713.927} C_VEL
LIN {X 0,Y 392.112,Z 616.73,A -85,B 0,C 180,E1 -11715.463,E2 -11715.463} C_VEL
LIN {X 0,Y 393.103,Z 604.612,A -85,B 0,C 180,E1 -11716.889,E2 -11716.889} C_VEL
LIN {X 0,Y 394.075,Z 592.573,A -85,B 0,C 180,E1 -11718.051,E2 -11718.051} C_VEL
LIN {X 0,Y 394.929,Z 580.144,A -85,B 0,C 180,E1 -11719.033,E2 -11719.033} C_VEL
LIN {X 0,Y 395.843,Z 566.023,A -85,B 0,C 180,E1 -11719.917,E2 -11719.917} C_VEL
LIN {X 0,Y 396.525,Z 551.691,A -85,B 0,C 180,E1 -11720.592,E2 -11720.592} C_VEL
LIN {X 0,Y 397.119,Z 537.188,A -85,B 0,C 180,E1 -11721.068,E2 -11721.068} C_VEL
LIN {X 0,Y 400.262,Z 426.947,A -85,B 0,C 180,E1 -11723.606,E2 -11723.606} C_VEL
LIN {X 0,Y 395.267,Z 397.796,A -85,B 0,C 180,E1 -11724.629,E2 -11724.629} C_VEL
LIN {X 0,Y 396.49,Z 384.195,A -85,B 0,C 180,E1 -11727.068,E2 -11727.068} C_VEL
LIN {X 0,Y 393.554,Z 371.136,A -85,B 0,C 180,E1 -11729.748,E2 -11729.748} C_VEL
LIN {X 0,Y 390.102,Z 356.724,A -85,B 0,C 180,E1 -11732.87,E2 -11732.87} C_VEL
LIN {X 0,Y 390.042,Z 356.527,A -85,B 0,C 180,E1 -11735.822,E2 -11735.822} C_VEL
LIN {X 0,Y 390.036,Z 356.525,A -85,B 0,C 180,E1 -11739.212,E2 -11739.212} C_VEL
LIN {X 0,Y 390.029,Z 356.508,A -85,B 0,C 180,E1 -11742.372,E2 -11742.372} C_VEL
LIN {X 0,Y 390.04,Z 356.526,A -85,B 0,C 180,E1 -11745.353,E2 -11745.353} C_VEL
LIN {X 0,Y 390.014,Z 356.523,A -85,B 0,C 180,E1 -11748.184,E2 -11748.184} C_VEL
LIN {X 0,Y 390.054,Z 356.514,A -85,B 0,C 180,E1 -11750.903,E2 -11750.903} C_VEL
LIN {X 0,Y 390.088,Z 356.695,A -85,B 0,C 180,E1 -11754.145,E2 -11754.145} C_VEL
LIN {X 0,Y 394.258,Z 371.151,A -85,B 0,C 180,E1 -11756.91,E2 -11756.91} C_VEL
LIN {X 0,Y 398.411,Z 387.567,A -85,B 0,C 180,E1 -11759.81,E2 -11759.81} C_VEL
LIN {X 0,Y 398.83,Z 391.578,A -85,B 0,C 180,E1 -11760.435,E2 -11760.435} C_VEL
LIN {X 0,Y 398.582,Z 396.96,A -85,B 0,C 180,E1 -11761.165,E2 -11761.165} C_VEL
LIN {X 0,Y 405.092,Z 430.443,A -85,B 0,C 180,E1 -11762.338,E2 -11762.338} C_VEL
LIN {X 0,Y 403.561,Z 512.999,A -85,B 0,C 180,E1 -11763.844,E2 -11763.844} C_VEL
LIN {X 0,Y 402.408,Z 564.843,A -85,B 0,C 180,E1 -11764.804,E2 -11764.804} C_VEL
LIN {X 0,Y 401.666,Z 579.703,A -85,B 0,C 180,E1 -11765.252,E2 -11765.252} C_VEL
LIN {X 0,Y 400.7,Z 593.855,A -85,B 0,C 180,E1 -11765.865,E2 -11765.865} C_VEL
LIN {X 0,Y 399.557,Z 608.072,A -85,B 0,C 180,E1 -11766.686,E2 -11766.686} C_VEL
LIN {X 0,Y 398.893,Z 614.699,A -85,B 0,C 180,E1 -11767.141,E2 -11767.141} C_VEL
LIN {X 0,Y 397.662,Z 619.985,A -85,B 0,C 180,E1 -11767.498,E2 -11767.498} C_VEL
LIN {X 0,Y 394.095,Z 628.343,A -85,B 0,C 180,E1 -11768.059,E2 -11768.059} C_VEL
LIN {X 0,Y 390.515,Z 636.47,A -85,B 0,C 180,E1 -11768.697,E2 -11768.697} C_VEL
LIN {X 0,Y 389.267,Z 641.207,A -85,B 0,C 180,E1 -11769.176,E2 -11769.176} C_VEL
LIN {X 0,Y 387.719,Z 653.027,A -85,B 0,C 180,E1 -11770.63,E2 -11770.63} C_VEL
LIN {X 0,Y 386.238,Z 664.01,A -85,B 0,C 180,E1 -11772.255,E2 -11772.255} C_VEL
LIN {X 0,Y 384.878,Z 674.357,A -85,B 0,C 180,E1 -11774.103,E2 -11774.103} C_VEL
LIN {X 0,Y 383.653,Z 683.733,A -85,B 0,C 180,E1 -11776.142,E2 -11776.142} C_VEL
LIN {X 0,Y 383.024,Z 690.125,A -85,B 0,C 180,E1 -11777.818,E2 -11777.818} C_VEL
LIN {X 0,Y 382.283,Z 696.752,A -85,B 0,C 180,E1 -11779.942,E2 -11779.942} C_VEL
LIN {X 0,Y 381.877,Z 701.94,A -85,B 0,C 180,E1 -11782.066,E2 -11782.066} C_VEL
LIN {X 0,Y 381.658,Z 705.367,A -85,B 0,C 180,E1 -11783.922,E2 -11783.922} C_VEL
LIN {X 0,Y 381.591,Z 707.862,A -85,B 0,C 180,E1 -11785.775,E2 -11785.775} C_VEL
LIN {X 0,Y 381.51,Z 709.624,A -85,B 0,C 180,E1 -11787.888,E2 -11787.888} C_VEL
LIN {X 0,Y 381.54,Z 710.235,A -85,B 0,C 180,E1 -11790,E2 -11790} C_VEL
LIN {X 0,Y 381.51,Z 709.665,A -85,B 0,C 180,E1 -11792.111,E2 -11792.111} C_VEL
LIN {X 0,Y 381.594,Z 707.96,A -85,B 0,C 180,E1 -11794.225,E2 -11794.225} C_VEL
LIN {X 0,Y 381.71,Z 705.085,A -85,B 0,C 180,E1 -11796.342,E2 -11796.342} C_VEL
LIN {X 0,Y 381.966,Z 700.973,A -85,B 0,C 180,E1 -11798.464,E2 -11798.464} C_VEL
LIN {X 0,Y 382.379,Z 695.513,A -85,B 0,C 180,E1 -11800.591,E2 -11800.591} C_VEL
LIN {X 0,Y 383.172,Z 688.56,A -85,B 0,C 180,E1 -11802.715,E2 -11802.715} C_VEL
LIN {X 0,Y 383.999,Z 681.238,A -85,B 0,C 180,E1 -11804.548,E2 -11804.548} C_VEL
LIN {X 0,Y 385.196,Z 672.151,A -85,B 0,C 180,E1 -11806.427,E2 -11806.427} C_VEL
LIN {X 0,Y 386.682,Z 661.314,A -85,B 0,C 180,E1 -11808.271,E2 -11808.271} C_VEL
LIN {X 0,Y 388.061,Z 650.452,A -85,B 0,C 180,E1 -11809.816,E2 -11809.816} C_VEL
LIN {X 0,Y 389.696,Z 637.98,A -85,B 0,C 180,E1 -11811.281,E2 -11811.281} C_VEL
LIN {X 0,Y 391.305,Z 624.509,A -85,B 0,C 180,E1 -11812.576,E2 -11812.576} C_VEL
LIN {X 0,Y 392.749,Z 611.337,A -85,B 0,C 180,E1 -11813.602,E2 -11813.602} C_VEL
LIN {X 0,Y 394.013,Z 596.941,A -85,B 0,C 180,E1 -11814.496,E2 -11814.496} C_VEL
LIN {X 0,Y 395.105,Z 581.678,A -85,B 0,C 180,E1 -11815.205,E2 -11815.205} C_VEL
LIN {X 0,Y 395.943,Z 565.926,A -85,B 0,C 180,E1 -11815.707,E2 -11815.707} C_VEL
LIN {X 0,Y 397.164,Z 516.173,A -85,B 0,C 180,E1 -11816.645,E2 -11816.645} C_VEL
LIN {X 0,Y 398.922,Z 432.14,A -85,B 0,C 180,E1 -11818.192,E2 -11818.192} C_VEL
LIN {X 0,Y 393.41,Z 403.333,A -85,B 0,C 180,E1 -11819.21,E2 -11819.21} C_VEL
LIN {X 0,Y 392.061,Z 396.697,A -85,B 0,C 180,E1 -11819.478,E2 -11819.478} C_VEL
LIN {X 0,Y 392.118,Z 391.458,A -85,B 0,C 180,E1 -11820.226,E2 -11820.226} C_VEL
LIN {X 0,Y 388.51,Z 376.423,A -85,B 0,C 180,E1 -11822.867,E2 -11822.867} C_VEL
LIN {X 0,Y 384.495,Z 362.444,A -85,B 0,C 180,E1 -11825.513,E2 -11825.513} C_VEL
LIN {X 0,Y 383.024,Z 357.569,A -85,B 0,C 180,E1 -11826.514,E2 -11826.514} C_VEL
LIN {X 0,Y 382.973,Z 357.39,A -85,B 0,C 180,E1 -11829.963,E2 -11829.963} C_VEL
LIN {X 0,Y 383.006,Z 357.397,A -85,B 0,C 180,E1 -11832.778,E2 -11832.778} C_VEL
LIN {X 0,Y 382.994,Z 357.402,A -85,B 0,C 180,E1 -11835.789,E2 -11835.789} C_VEL
LIN {X 0,Y 382.961,Z 357.408,A -85,B 0,C 180,E1 -11838.8,E2 -11838.8} C_VEL
LIN {X 0,Y 382.992,Z 357.404,A -85,B 0,C 180,E1 -11842.098,E2 -11842.098} C_VEL
LIN {X 0,Y 383.012,Z 357.394,A -85,B 0,C 180,E1 -11845.331,E2 -11845.331} C_VEL
LIN {X 0,Y 382.982,Z 357.394,A -85,B 0,C 180,E1 -11849.081,E2 -11849.081} C_VEL
LIN {X 0,Y 382.991,Z 357.389,A -85,B 0,C 180,E1 -11852.693,E2 -11852.693} C_VEL
LIN {X 0,Y 383.01,Z 357.396,A -85,B 0,C 180,E1 -11856.191,E2 -11856.191} C_VEL
LIN {X 0,Y 383.056,Z 357.392,A -85,B 0,C 180,E1 -11859.598,E2 -11859.598} C_VEL
LIN {X 0,Y 383.094,Z 357.375,A -85,B 0,C 180,E1 -11862.931,E2 -11862.931} C_VEL
LIN {X 0,Y 383.126,Z 357.384,A -85,B 0,C 180,E1 -11866.464,E2 -11866.464} C_VEL
LIN {X 0,Y 383.143,Z 357.377,A -85,B 0,C 180,E1 -11870.498,E2 -11870.498} C_VEL
LIN {X 0,Y 383.274,Z 357.358,A -85,B 0,C 180,E1 -11873.683,E2 -11873.683} C_VEL
LIN {X 0,Y 383.379,Z 357.355,A -85,B 0,C 180,E1 -11877.899,E2 -11877.899} C_VEL
LIN {X 0,Y 383.516,Z 357.328,A -85,B 0,C 180,E1 -11880,E2 -11880} C_VEL
LIN {X 0,Y 383.24,Z 357.363,A -85,B 0,C 180,E1 -11883.154,E2 -11883.154} C_VEL
LIN {X 0,Y 383.256,Z 357.361,A -85,B 0,C 180,E1 -11886.317,E2 -11886.317} C_VEL
LIN {X 0,Y 383.144,Z 357.377,A -85,B 0,C 180,E1 -11889.502,E2 -11889.502} C_VEL
LIN {X 0,Y 383.137,Z 357.375,A -85,B 0,C 180,E1 -11892.716,E2 -11892.716} C_VEL
LIN {X 0,Y 383.081,Z 357.389,A -85,B 0,C 180,E1 -11895.973,E2 -11895.973} C_VEL
LIN {X 0,Y 383.059,Z 357.379,A -85,B 0,C 180,E1 -11899.284,E2 -11899.284} C_VEL
LIN {X 0,Y 383.013,Z 357.4,A -85,B 0,C 180,E1 -11902.664,E2 -11902.664} C_VEL
LIN {X 0,Y 383.08,Z 357.386,A -85,B 0,C 180,E1 -11906.123,E2 -11906.123} C_VEL
LIN {X 0,Y 383.04,Z 357.396,A -85,B 0,C 180,E1 -11908.493,E2 -11908.493} C_VEL
LIN {X 0,Y 383.009,Z 357.4,A -85,B 0,C 180,E1 -11912.15,E2 -11912.15} C_VEL
LIN {X 0,Y 383.018,Z 357.389,A -85,B 0,C 180,E1 -11914.668,E2 -11914.668} C_VEL
LIN {X 0,Y 382.998,Z 357.394,A -85,B 0,C 180,E1 -11917.903,E2 -11917.903} C_VEL
LIN {X 0,Y 382.984,Z 357.371,A -85,B 0,C 180,E1 -11921.347,E2 -11921.347} C_VEL
LIN {X 0,Y 382.998,Z 357.403,A -85,B 0,C 180,E1 -11924.304,E2 -11924.304} C_VEL
LIN {X 0,Y 383.009,Z 357.372,A -85,B 0,C 180,E1 -11927.24,E2 -11927.24} C_VEL
LIN {X 0,Y 383.015,Z 357.401,A -85,B 0,C 180,E1 -11930.413,E2 -11930.413} C_VEL
LIN {X 0,Y 383.041,Z 357.527,A -85,B 0,C 180,E1 -11934.33,E2 -11934.33} C_VEL
LIN {X 0,Y 387.092,Z 372.591,A -85,B 0,C 180,E1 -11937.307,E2 -11937.307} C_VEL
LIN {X 0,Y 391.407,Z 389.362,A -85,B 0,C 180,E1 -11940.41,E2 -11940.41} C_VEL
LIN {X 0,Y 391.773,Z 391.46,A -85,B 0,C 180,E1 -11940.716,E2 -11940.716} C_VEL
LIN {X 0,Y 397.918,Z 427.566,A -85,B 0,C 180,E1 -11941.951,E2 -11941.951} C_VEL
LIN {X 0,Y 398.273,Z 431.461,A -85,B 0,C 180,E1 -11942.056,E2 -11942.056} C_VEL
LIN {X 0,Y 395.358,Z 565.665,A -85,B 0,C 180,E1 -11944.535,E2 -11944.535} C_VEL
LIN {X 0,Y 394.526,Z 581.432,A -85,B 0,C 180,E1 -11945.038,E2 -11945.038} C_VEL
LIN {X 0,Y 393.424,Z 596.535,A -85,B 0,C 180,E1 -11945.741,E2 -11945.741} C_VEL
LIN {X 0,Y 392.222,Z 611.063,A -85,B 0,C 180,E1 -11946.651,E2 -11946.651} C_VEL
LIN {X 0,Y 390.769,Z 624.148,A -85,B 0,C 180,E1 -11947.67,E2 -11947.67} C_VEL
LIN {X 0,Y 389.234,Z 637.526,A -85,B 0,C 180,E1 -11948.97,E2 -11948.97} C_VEL
LIN {X 0,Y 387.798,Z 649.16,A -85,B 0,C 180,E1 -11950.34,E2 -11950.34} C_VEL
LIN {X 0,Y 386.294,Z 660.729,A -85,B 0,C 180,E1 -11951.984,E2 -11951.984} C_VEL
LIN {X 0,Y 384.865,Z 671.445,A -85,B 0,C 180,E1 -11953.831,E2 -11953.831} C_VEL
LIN {X 0,Y 383.79,Z 680.343,A -85,B 0,C 180,E1 -11955.687,E2 -11955.687} C_VEL
LIN {X 0,Y 382.916,Z 688.653,A -85,B 0,C 180,E1 -11957.815,E2 -11957.815} C_VEL
LIN {X 0,Y 382.235,Z 695.313,A -85,B 0,C 180,E1 -11959.941,E2 -11959.941} C_VEL
LIN {X 0,Y 381.871,Z 700.513,A -85,B 0,C 180,E1 -11962.066,E2 -11962.066} C_VEL
LIN {X 0,Y 381.686,Z 703.872,A -85,B 0,C 180,E1 -11963.88,E2 -11963.88} C_VEL
LIN {X 0,Y 381.596,Z 706.423,A -85,B 0,C 180,E1 -11965.775,E2 -11965.775} C_VEL
LIN {X 0,Y 381.562,Z 708.168,A -85,B 0,C 180,E1 -11967.889,E2 -11967.889} C_VEL
LIN {X 0,Y 381.538,Z 708.763,A -85,B 0,C 180,E1 -11970,E2 -11970} C_VEL
LIN {X 0,Y 381.564,Z 708.167,A -85,B 0,C 180,E1 -11972.111,E2 -11972.111} C_VEL
LIN {X 0,Y 381.595,Z 706.42,A -85,B 0,C 180,E1 -11974.225,E2 -11974.225} C_VEL
LIN {X 0,Y 381.7,Z 703.487,A -85,B 0,C 180,E1 -11976.343,E2 -11976.343} C_VEL
LIN {X 0,Y 381.958,Z 699.301,A -85,B 0,C 180,E1 -11978.465,E2 -11978.465} C_VEL
LIN {X 0,Y 382.344,Z 693.758,A -85,B 0,C 180,E1 -11980.592,E2 -11980.592} C_VEL
LIN {X 0,Y 383.085,Z 686.701,A -85,B 0,C 180,E1 -11982.718,E2 -11982.718} C_VEL
LIN {X 0,Y 383.959,Z 679.126,A -85,B 0,C 180,E1 -11984.577,E2 -11984.577} C_VEL
LIN {X 0,Y 385.086,Z 669.987,A -85,B 0,C 180,E1 -11986.432,E2 -11986.432} C_VEL
LIN {X 0,Y 386.274,Z 660.675,A -85,B 0,C 180,E1 -11988.017,E2 -11988.017} C_VEL
LIN {X 0,Y 387.824,Z 648.998,A -85,B 0,C 180,E1 -11989.67,E2 -11989.67} C_VEL
LIN {X 0,Y 389.382,Z 636.203,A -85,B 0,C 180,E1 -11991.161,E2 -11991.161} C_VEL
LIN {X 0,Y 390.975,Z 622.499,A -85,B 0,C 180,E1 -11992.457,E2 -11992.457} C_VEL
LIN {X 0,Y 392.431,Z 608.98,A -85,B 0,C 180,E1 -11993.483,E2 -11993.483} C_VEL
LIN {X 0,Y 393.598,Z 595.293,A -85,B 0,C 180,E1 -11994.311,E2 -11994.311} C_VEL
LIN {X 0,Y 394.62,Z 580.44,A -85,B 0,C 180,E1 -11994.987,E2 -11994.987} C_VEL
LIN {X 0,Y 395.381,Z 565.252,A -85,B 0,C 180,E1 -11995.464,E2 -11995.464} C_VEL
LIN {X 0,Y 396.196,Z 542.81,A -85,B 0,C 180,E1 -11995.972,E2 -11995.972} C_VEL
LIN {X 0,Y 399.73,Z 474.843,A -85,B 0,C 180,E1 -11997.733,E2 -11997.733} C_VEL
LIN {X 0,Y 402.477,Z 430.32,A -85,B 0,C 180,E1 -11998.963,E2 -11998.963} C_VEL
LIN {X 0,Y 400.817,Z 416.581,A -85,B 0,C 180,E1 -11999.681,E2 -11999.681} C_VEL
LIN {X 0,Y 398.539,Z 404.237,A -85,B 0,C 180,E1 -12000.472,E2 -12000.472} C_VEL
LIN {X 0,Y 397.659,Z 401.236,A -85,B 0,C 180,E1 -12000.72,E2 -12000.72} C_VEL
LIN {X 0,Y 396.629,Z 398.729,A -85,B 0,C 180,E1 -12001.027,E2 -12001.027} C_VEL
LIN {X 0,Y 395.26,Z 392.173,A -85,B 0,C 180,E1 -12002.799,E2 -12002.799} C_VEL
LIN {X 0,Y 393.621,Z 385.806,A -85,B 0,C 180,E1 -12004.845,E2 -12004.845} C_VEL
LIN {X 0,Y 392.058,Z 380.7,A -85,B 0,C 180,E1 -12006.84,E2 -12006.84} C_VEL
LIN {X 0,Y 390.591,Z 376.304,A -85,B 0,C 180,E1 -12009.033,E2 -12009.033} C_VEL
LIN {X 0,Y 389.656,Z 373.784,A -85,B 0,C 180,E1 -12010.753,E2 -12010.753} C_VEL
LIN {X 0,Y 389.119,Z 372.123,A -85,B 0,C 180,E1 -12012.225,E2 -12012.225} C_VEL
LIN {X 0,Y 388.66,Z 371.093,A -85,B 0,C 180,E1 -12013.672,E2 -12013.672} C_VEL
LIN {X 0,Y 388.37,Z 370.626,A -85,B 0,C 180,E1 -12015.11,E2 -12015.11} C_VEL
LIN {X 0,Y 388.518,Z 370.946,A -85,B 0,C 180,E1 -12017.873,E2 -12017.873} C_VEL
LIN {X 0,Y 388.868,Z 371.901,A -85,B 0,C 180,E1 -12019.411,E2 -12019.411} C_VEL
LIN {X 0,Y 389.964,Z 375.095,A -85,B 0,C 180,E1 -12022.211,E2 -12022.211} C_VEL
LIN {X 0,Y 390.917,Z 378.076,A -85,B 0,C 180,E1 -12024.001,E2 -12024.001} C_VEL
LIN {X 0,Y 392.312,Z 382.917,A -85,B 0,C 180,E1 -12026.266,E2 -12026.266} C_VEL
LIN {X 0,Y 393.931,Z 389.858,A -85,B 0,C 180,E1 -12028.843,E2 -12028.843} C_VEL
LIN {X 0,Y 395.349,Z 397.901,A -85,B 0,C 180,E1 -12031.317,E2 -12031.317} C_VEL
LIN {X 0,Y 395.545,Z 399.535,A -85,B 0,C 180,E1 -12031.618,E2 -12031.618} C_VEL
LIN {X 0,Y 398.576,Z 411.487,A -85,B 0,C 180,E1 -12032.613,E2 -12032.613} C_VEL
LIN {X 0,Y 400.847,Z 423.054,A -85,B 0,C 180,E1 -12033.403,E2 -12033.403} C_VEL
LIN {X 0,Y 402.157,Z 431.893,A -85,B 0,C 180,E1 -12033.923,E2 -12033.923} C_VEL
LIN {X 0,Y 396.615,Z 512.117,A -85,B 0,C 180,E1 -12036.296,E2 -12036.296} C_VEL
LIN {X 0,Y 394.662,Z 546.32,A -85,B 0,C 180,E1 -12037.316,E2 -12037.316} C_VEL
LIN {X 0,Y 393.533,Z 561.449,A -85,B 0,C 180,E1 -12037.974,E2 -12037.974} C_VEL
LIN {X 0,Y 392.3,Z 576.218,A -85,B 0,C 180,E1 -12038.849,E2 -12038.849} C_VEL
LIN {X 0,Y 390.878,Z 590.03,A -85,B 0,C 180,E1 -12039.894,E2 -12039.894} C_VEL
LIN {X 0,Y 389.309,Z 603.62,A -85,B 0,C 180,E1 -12041.175,E2 -12041.175} C_VEL
LIN {X 0,Y 387.933,Z 615.88,A -85,B 0,C 180,E1 -12042.607,E2 -12042.607} C_VEL
LIN {X 0,Y 386.578,Z 626.843,A -85,B 0,C 180,E1 -12044.175,E2 -12044.175} C_VEL
LIN {X 0,Y 385.333,Z 635.978,A -85,B 0,C 180,E1 -12045.746,E2 -12045.746} C_VEL
LIN {X 0,Y 384.248,Z 644.729,A -85,B 0,C 180,E1 -12047.59,E2 -12047.59} C_VEL
LIN {X 0,Y 383.417,Z 651.794,A -85,B 0,C 180,E1 -12049.438,E2 -12049.438} C_VEL
LIN {X 0,Y 382.875,Z 656.688,A -85,B 0,C 180,E1 -12051.024,E2 -12051.024} C_VEL
LIN {X 0,Y 382.363,Z 661.425,A -85,B 0,C 180,E1 -12053.001,E2 -12053.001} C_VEL
LIN {X 0,Y 382,Z 664.444,A -85,B 0,C 180,E1 -12054.722,E2 -12054.722} C_VEL
LIN {X 0,Y 381.953,Z 666.75,A -85,B 0,C 180,E1 -12056.836,E2 -12056.836} C_VEL
LIN {X 0,Y 381.716,Z 667.64,A -85,B 0,C 180,E1 -12058.945,E2 -12058.945} C_VEL
LIN {X 0,Y 381.705,Z 667.088,A -85,B 0,C 180,E1 -12061.055,E2 -12061.055} C_VEL
LIN {X 0,Y 381.771,Z 666.274,A -85,B 0,C 180,E1 -12062.11,E2 -12062.11} C_VEL
LIN {X 0,Y 381.772,Z 663.56,A -85,B 0,C 180,E1 -12064.223,E2 -12064.223} C_VEL
LIN {X 0,Y 381.979,Z 660.492,A -85,B 0,C 180,E1 -12065.808,E2 -12065.808} C_VEL
LIN {X 0,Y 382.149,Z 656.551,A -85,B 0,C 180,E1 -12067.397,E2 -12067.397} C_VEL
LIN {X 0,Y 382.408,Z 651.628,A -85,B 0,C 180,E1 -12068.987,E2 -12068.987} C_VEL
LIN {X 0,Y 382.93,Z 644.479,A -85,B 0,C 180,E1 -12070.843,E2 -12070.843} C_VEL
LIN {X 0,Y 383.544,Z 636.995,A -85,B 0,C 180,E1 -12072.434,E2 -12072.434} C_VEL
LIN {X 0,Y 384.285,Z 627.768,A -85,B 0,C 180,E1 -12074.062,E2 -12074.062} C_VEL
LIN {X 0,Y 385.116,Z 617.118,A -85,B 0,C 180,E1 -12075.615,E2 -12075.615} C_VEL
LIN {X 0,Y 386.141,Z 605.008,A -85,B 0,C 180,E1 -12077.067,E2 -12077.067} C_VEL
LIN {X 0,Y 387.142,Z 592.991,A -85,B 0,C 180,E1 -12078.249,E2 -12078.249} C_VEL
LIN {X 0,Y 388.119,Z 579.455,A -85,B 0,C 180,E1 -12079.333,E2 -12079.333} C_VEL
LIN {X 0,Y 388.993,Z 565.363,A -85,B 0,C 180,E1 -12080.215,E2 -12080.215} C_VEL
LIN {X 0,Y 389.73,Z 550.792,A -85,B 0,C 180,E1 -12080.899,E2 -12080.899} C_VEL
LIN {X 0,Y 390.33,Z 535.887,A -85,B 0,C 180,E1 -12081.384,E2 -12081.384} C_VEL
LIN {X 0,Y 393.511,Z 427.368,A -85,B 0,C 180,E1 -12083.952,E2 -12083.952} C_VEL
LIN {X 0,Y 388.508,Z 397.87,A -85,B 0,C 180,E1 -12085.015,E2 -12085.015} C_VEL
LIN {X 0,Y 389.573,Z 385.31,A -85,B 0,C 180,E1 -12087.298,E2 -12087.298} C_VEL
LIN {X 0,Y 386.238,Z 370.82,A -85,B 0,C 180,E1 -12090.327,E2 -12090.327} C_VEL
LIN {X 0,Y 383.072,Z 357.55,A -85,B 0,C 180,E1 -12093.275,E2 -12093.275} C_VEL
LIN {X 0,Y 383.021,Z 357.402,A -85,B 0,C 180,E1 -12096.162,E2 -12096.162} C_VEL
LIN {X 0,Y 382.985,Z 357.405,A -85,B 0,C 180,E1 -12099.581,E2 -12099.581} C_VEL
LIN {X 0,Y 383.007,Z 357.382,A -85,B 0,C 180,E1 -12102.779,E2 -12102.779} C_VEL
LIN {X 0,Y 382.99,Z 357.397,A -85,B 0,C 180,E1 -12105.788,E2 -12105.788} C_VEL
LIN {X 0,Y 382.962,Z 357.408,A -85,B 0,C 180,E1 -12108.801,E2 -12108.801} C_VEL
LIN {X 0,Y 382.991,Z 357.404,A -85,B 0,C 180,E1 -12112.098,E2 -12112.098} C_VEL
LIN {X 0,Y 383.042,Z 357.572,A -85,B 0,C 180,E1 -12113.598,E2 -12113.598} C_VEL
LIN {X 0,Y 387.019,Z 370.973,A -85,B 0,C 180,E1 -12116.225,E2 -12116.225} C_VEL
LIN {X 0,Y 390.262,Z 383.544,A -85,B 0,C 180,E1 -12118.517,E2 -12118.517} C_VEL
LIN {X 0,Y 392.176,Z 391.504,A -85,B 0,C 180,E1 -12119.882,E2 -12119.882} C_VEL
LIN {X 0,Y 392.052,Z 396.736,A -85,B 0,C 180,E1 -12120.629,E2 -12120.629} C_VEL
LIN {X 0,Y 397.673,Z 425.407,A -85,B 0,C 180,E1 -12121.678,E2 -12121.678} C_VEL
LIN {X 0,Y 398.897,Z 433.039,A -85,B 0,C 180,E1 -12121.925,E2 -12121.925} C_VEL
LIN {X 0,Y 396.246,Z 555.682,A -85,B 0,C 180,E1 -12124.173,E2 -12124.173} C_VEL
LIN {X 0,Y 395.662,Z 571.758,A -85,B 0,C 180,E1 -12124.555,E2 -12124.555} C_VEL
LIN {X 0,Y 394.716,Z 587.081,A -85,B 0,C 180,E1 -12125.122,E2 -12125.122} C_VEL
LIN {X 0,Y 393.532,Z 601.92,A -85,B 0,C 180,E1 -12125.888,E2 -12125.888} C_VEL
LIN {X 0,Y 392.257,Z 615.335,A -85,B 0,C 180,E1 -12126.786,E2 -12126.786} C_VEL
LIN {X 0,Y 390.718,Z 629.197,A -85,B 0,C 180,E1 -12127.945,E2 -12127.945} C_VEL
LIN {X 0,Y 389.267,Z 641.207,A -85,B 0,C 180,E1 -12129.176,E2 -12129.176} C_VEL
LIN {X 0,Y 387.984,Z 645.904,A -85,B 0,C 180,E1 -12129.681,E2 -12129.681} C_VEL
LIN {X 0,Y 384.241,Z 653.297,A -85,B 0,C 180,E1 -12130.488,E2 -12130.488} C_VEL
LIN {X 0,Y 380.553,Z 660.359,A -85,B 0,C 180,E1 -12131.371,E2 -12131.371} C_VEL
LIN {X 0,Y 379.364,Z 664.394,A -85,B 0,C 180,E1 -12131.992,E2 -12131.992} C_VEL
LIN {X 0,Y 378.005,Z 674.341,A -85,B 0,C 180,E1 -12133.806,E2 -12133.806} C_VEL
LIN {X 0,Y 376.82,Z 682.947,A -85,B 0,C 180,E1 -12135.692,E2 -12135.692} C_VEL
LIN {X 0,Y 376.026,Z 690.11,A -85,B 0,C 180,E1 -12137.588,E2 -12137.588} C_VEL
LIN {X 0,Y 375.257,Z 696.738,A -85,B 0,C 180,E1 -12139.751,E2 -12139.751} C_VEL
LIN {X 0,Y 374.822,Z 701.926,A -85,B 0,C 180,E1 -12141.916,E2 -12141.916} C_VEL
LIN {X 0,Y 374.553,Z 705.631,A -85,B 0,C 180,E1 -12143.976,E2 -12143.976} C_VEL
LIN {X 0,Y 374.496,Z 707.849,A -85,B 0,C 180,E1 -12145.695,E2 -12145.695} C_VEL
LIN {X 0,Y 374.409,Z 709.61,A -85,B 0,C 180,E1 -12147.848,E2 -12147.848} C_VEL
LIN {X 0,Y 374.44,Z 710.221,A -85,B 0,C 180,E1 -12150,E2 -12150} C_VEL
LIN {X 0,Y 374.41,Z 709.651,A -85,B 0,C 180,E1 -12152.151,E2 -12152.151} C_VEL
LIN {X 0,Y 374.5,Z 707.945,A -85,B 0,C 180,E1 -12154.305,E2 -12154.305} C_VEL
LIN {X 0,Y 374.628,Z 705.07,A -85,B 0,C 180,E1 -12156.463,E2 -12156.463} C_VEL
LIN {X 0,Y 374.919,Z 700.957,A -85,B 0,C 180,E1 -12158.625,E2 -12158.625} C_VEL
LIN {X 0,Y 375.349,Z 695.496,A -85,B 0,C 180,E1 -12160.792,E2 -12160.792} C_VEL
LIN {X 0,Y 376.174,Z 688.542,A -85,B 0,C 180,E1 -12162.955,E2 -12162.955} C_VEL
LIN {X 0,Y 377.072,Z 681.097,A -85,B 0,C 180,E1 -12164.849,E2 -12164.849} C_VEL
LIN {X 0,Y 378.318,Z 672.13,A -85,B 0,C 180,E1 -12166.735,E2 -12166.735} C_VEL
LIN {X 0,Y 379.646,Z 662.965,A -85,B 0,C 180,E1 -12168.343,E2 -12168.343} C_VEL
LIN {X 0,Y 381.114,Z 651.961,A -85,B 0,C 180,E1 -12169.973,E2 -12169.973} C_VEL
LIN {X 0,Y 382.694,Z 640.318,A -85,B 0,C 180,E1 -12171.407,E2 -12171.407} C_VEL
LIN {X 0,Y 384.359,Z 627.379,A -85,B 0,C 180,E1 -12172.723,E2 -12172.723} C_VEL
LIN {X 0,Y 385.86,Z 614.802,A -85,B 0,C 180,E1 -12173.765,E2 -12173.765} C_VEL
LIN {X 0,Y 387.177,Z 601.256,A -85,B 0,C 180,E1 -12174.676,E2 -12174.676} C_VEL
LIN {X 0,Y 388.329,Z 585.949,A -85,B 0,C 180,E1 -12175.471,E2 -12175.471} C_VEL
LIN {X 0,Y 389.36,Z 570.461,A -85,B 0,C 180,E1 -12176.03,E2 -12176.03} C_VEL
LIN {X 0,Y 389.962,Z 553.475,A -85,B 0,C 180,E1 -12176.418,E2 -12176.418} C_VEL
LIN {X 0,Y 392.663,Z 433.305,A -85,B 0,C 180,E1 -12178.655,E2 -12178.655} C_VEL
LIN {X 0,Y 387.129,Z 404.262,A -85,B 0,C 180,E1 -12179.708,E2 -12179.708} C_VEL
LIN {X 0,Y 385.591,Z 396.507,A -85,B 0,C 180,E1 -12180.031,E2 -12180.031} C_VEL
LIN {X 0,Y 385.401,Z 393.025,A -85,B 0,C 180,E1 -12180.55,E2 -12180.55} C_VEL
LIN {X 0,Y 381.877,Z 378.547,A -85,B 0,C 180,E1 -12183.137,E2 -12183.137} C_VEL
LIN {X 0,Y 378.001,Z 365.023,A -85,B 0,C 180,E1 -12185.714,E2 -12185.714} C_VEL
LIN {X 0,Y 375.982,Z 358.492,A -85,B 0,C 180,E1 -12187.073,E2 -12187.073} C_VEL
LIN {X 0,Y 375.937,Z 358.266,A -85,B 0,C 180,E1 -12189.961,E2 -12189.961} C_VEL
LIN {X 0,Y 375.928,Z 358.286,A -85,B 0,C 180,E1 -12193.766,E2 -12193.766} C_VEL
LIN {X 0,Y 375.934,Z 358.284,A -85,B 0,C 180,E1 -12196.811,E2 -12196.811} C_VEL
LIN {X 0,Y 375.933,Z 358.277,A -85,B 0,C 180,E1 -12200.534,E2 -12200.534} C_VEL
LIN {X 0,Y 375.957,Z 358.277,A -85,B 0,C 180,E1 -12203.497,E2 -12203.497} C_VEL
LIN {X 0,Y 375.958,Z 358.279,A -85,B 0,C 180,E1 -12205.888,E2 -12205.888} C_VEL
LIN {X 0,Y 375.962,Z 358.274,A -85,B 0,C 180,E1 -12209.687,E2 -12209.687} C_VEL
LIN {X 0,Y 375.933,Z 358.271,A -85,B 0,C 180,E1 -12212.136,E2 -12212.136} C_VEL
LIN {X 0,Y 375.959,Z 358.279,A -85,B 0,C 180,E1 -12215.716,E2 -12215.716} C_VEL
LIN {X 0,Y 375.999,Z 358.266,A -85,B 0,C 180,E1 -12219.198,E2 -12219.198} C_VEL
LIN {X 0,Y 376.033,Z 358.256,A -85,B 0,C 180,E1 -12222.6,E2 -12222.6} C_VEL
LIN {X 0,Y 376.09,Z 358.261,A -85,B 0,C 180,E1 -12226.342,E2 -12226.342} C_VEL
LIN {X 0,Y 376.113,Z 358.252,A -85,B 0,C 180,E1 -12230.318,E2 -12230.318} C_VEL
LIN {X 0,Y 376.231,Z 358.237,A -85,B 0,C 180,E1 -12233.565,E2 -12233.565} C_VEL
LIN {X 0,Y 376.344,Z 358.231,A -85,B 0,C 180,E1 -12237.859,E2 -12237.859} C_VEL
LIN {X 0,Y 376.486,Z 358.203,A -85,B 0,C 180,E1 -12240,E2 -12240} C_VEL
LIN {X 0,Y 376.35,Z 358.214,A -85,B 0,C 180,E1 -12242.14,E2 -12242.14} C_VEL
LIN {X 0,Y 376.214,Z 358.238,A -85,B 0,C 180,E1 -12246.435,E2 -12246.435} C_VEL
LIN {X 0,Y 376.114,Z 358.255,A -85,B 0,C 180,E1 -12249.681,E2 -12249.681} C_VEL
LIN {X 0,Y 376.09,Z 358.243,A -85,B 0,C 180,E1 -12253.658,E2 -12253.658} C_VEL
LIN {X 0,Y 376.032,Z 358.268,A -85,B 0,C 180,E1 -12257.4,E2 -12257.4} C_VEL
LIN {X 0,Y 375.978,Z 358.266,A -85,B 0,C 180,E1 -12260.832,E2 -12260.832} C_VEL
LIN {X 0,Y 375.994,Z 358.265,A -85,B 0,C 180,E1 -12264.281,E2 -12264.281} C_VEL
LIN {X 0,Y 376.02,Z 358.267,A -85,B 0,C 180,E1 -12266.652,E2 -12266.652} C_VEL
LIN {X 0,Y 375.97,Z 358.269,A -85,B 0,C 180,E1 -12269.079,E2 -12269.079} C_VEL
LIN {X 0,Y 375.949,Z 358.282,A -85,B 0,C 180,E1 -12272.828,E2 -12272.828} C_VEL
LIN {X 0,Y 375.957,Z 358.275,A -85,B 0,C 180,E1 -12275.415,E2 -12275.415} C_VEL
LIN {X 0,Y 375.972,Z 358.26,A -85,B 0,C 180,E1 -12278.27,E2 -12278.27} C_VEL
LIN {X 0,Y 375.934,Z 358.252,A -85,B 0,C 180,E1 -12281.601,E2 -12281.601} C_VEL
LIN {X 0,Y 375.927,Z 358.267,A -85,B 0,C 180,E1 -12285.268,E2 -12285.268} C_VEL
LIN {X 0,Y 375.934,Z 358.27,A -85,B 0,C 180,E1 -12288.399,E2 -12288.399} C_VEL
LIN {X 0,Y 375.974,Z 358.278,A -85,B 0,C 180,E1 -12291.729,E2 -12291.729} C_VEL
LIN {X 0,Y 376.019,Z 358.475,A -85,B 0,C 180,E1 -12293.932,E2 -12293.932} C_VEL
LIN {X 0,Y 380.594,Z 375.524,A -85,B 0,C 180,E1 -12297.336,E2 -12297.336} C_VEL
LIN {X 0,Y 384.308,Z 389.974,A -85,B 0,C 180,E1 -12300.015,E2 -12300.015} C_VEL
LIN {X 0,Y 385.825,Z 393.976,A -85,B 0,C 180,E1 -12300.282,E2 -12300.282} C_VEL
LIN {X 0,Y 391.969,Z 430.523,A -85,B 0,C 180,E1 -12301.544,E2 -12301.544} C_VEL
LIN {X 0,Y 389.051,Z 564.355,A -85,B 0,C 180,E1 -12304.056,E2 -12304.056} C_VEL
LIN {X 0,Y 388.189,Z 579.902,A -85,B 0,C 180,E1 -12304.534,E2 -12304.534} C_VEL
LIN {X 0,Y 387.067,Z 595.421,A -85,B 0,C 180,E1 -12305.245,E2 -12305.245} C_VEL
LIN {X 0,Y 385.886,Z 609.504,A -85,B 0,C 180,E1 -12306.12,E2 -12306.12} C_VEL
LIN {X 0,Y 384.372,Z 622.644,A -85,B 0,C 180,E1 -12307.136,E2 -12307.136} C_VEL
LIN {X 0,Y 382.747,Z 636.332,A -85,B 0,C 180,E1 -12308.455,E2 -12308.455} C_VEL
LIN {X 0,Y 381.12,Z 648.859,A -85,B 0,C 180,E1 -12309.937,E2 -12309.937} C_VEL
LIN {X 0,Y 379.525,Z 660.752,A -85,B 0,C 180,E1 -12311.651,E2 -12311.651} C_VEL
LIN {X 0,Y 378.206,Z 670.057,A -85,B 0,C 180,E1 -12313.26,E2 -12313.26} C_VEL
LIN {X 0,Y 376.997,Z 679.18,A -85,B 0,C 180,E1 -12315.148,E2 -12315.148} C_VEL
LIN {X 0,Y 376.06,Z 686.744,A -85,B 0,C 180,E1 -12317.041,E2 -12317.041} C_VEL
LIN {X 0,Y 375.311,Z 693.799,A -85,B 0,C 180,E1 -12319.207,E2 -12319.207} C_VEL
LIN {X 0,Y 374.91,Z 699.338,A -85,B 0,C 180,E1 -12321.375,E2 -12321.375} C_VEL
LIN {X 0,Y 374.622,Z 703.513,A -85,B 0,C 180,E1 -12323.537,E2 -12323.537} C_VEL
LIN {X 0,Y 374.501,Z 706.437,A -85,B 0,C 180,E1 -12325.695,E2 -12325.695} C_VEL
LIN {X 0,Y 374.459,Z 708.182,A -85,B 0,C 180,E1 -12327.849,E2 -12327.849} C_VEL
LIN {X 0,Y 374.439,Z 708.777,A -85,B 0,C 180,E1 -12330,E2 -12330} C_VEL
LIN {X 0,Y 374.462,Z 708.181,A -85,B 0,C 180,E1 -12332.151,E2 -12332.151} C_VEL
LIN {X 0,Y 374.501,Z 706.433,A -85,B 0,C 180,E1 -12334.305,E2 -12334.305} C_VEL
LIN {X 0,Y 374.622,Z 703.501,A -85,B 0,C 180,E1 -12336.463,E2 -12336.463} C_VEL
LIN {X 0,Y 374.91,Z 699.315,A -85,B 0,C 180,E1 -12338.625,E2 -12338.625} C_VEL
LIN {X 0,Y 375.314,Z 693.773,A -85,B 0,C 180,E1 -12340.793,E2 -12340.793} C_VEL
LIN {X 0,Y 375.928,Z 688.645,A -85,B 0,C 180,E1 -12342.415,E2 -12342.415} C_VEL
LIN {X 0,Y 376.878,Z 680.327,A -85,B 0,C 180,E1 -12344.581,E2 -12344.581} C_VEL
LIN {X 0,Y 378.029,Z 671.417,A -85,B 0,C 180,E1 -12346.47,E2 -12346.47} C_VEL
LIN {X 0,Y 379.226,Z 662.314,A -85,B 0,C 180,E1 -12348.085,E2 -12348.085} C_VEL
LIN {X 0,Y 380.738,Z 651.382,A -85,B 0,C 180,E1 -12349.712,E2 -12349.712} C_VEL
LIN {X 0,Y 382.247,Z 639.789,A -85,B 0,C 180,E1 -12351.151,E2 -12351.151} C_VEL
LIN {X 0,Y 383.893,Z 626.907,A -85,B 0,C 180,E1 -12352.468,E2 -12352.468} C_VEL
LIN {X 0,Y 385.313,Z 614.393,A -85,B 0,C 180,E1 -12353.515,E2 -12353.515} C_VEL
LIN {X 0,Y 386.73,Z 599.775,A -85,B 0,C 180,E1 -12354.491,E2 -12354.491} C_VEL
LIN {X 0,Y 387.912,Z 584.332,A -85,B 0,C 180,E1 -12355.27,E2 -12355.27} C_VEL
LIN {X 0,Y 388.808,Z 568.813,A -85,B 0,C 180,E1 -12355.818,E2 -12355.818} C_VEL
LIN {X 0,Y 394.651,Z 467.758,A -85,B 0,C 180,E1 -12358.557,E2 -12358.557} C_VEL
LIN {X 0,Y 397.05,Z 431.519,A -85,B 0,C 180,E1 -12359.602,E2 -12359.602} C_VEL
LIN {X 0,Y 395.474,Z 417.799,A -85,B 0,C 180,E1 -12360.356,E2 -12360.356} C_VEL
LIN {X 0,Y 393.341,Z 405.938,A -85,B 0,C 180,E1 -12361.168,E2 -12361.168} C_VEL
LIN {X 0,Y 389.945,Z 398.959,A -85,B 0,C 180,E1 -12362.057,E2 -12362.057} C_VEL
LIN {X 0,Y 388.384,Z 392.152,A -85,B 0,C 180,E1 -12364.122,E2 -12364.122} C_VEL
LIN {X 0,Y 386.752,Z 386.2,A -85,B 0,C 180,E1 -12366.342,E2 -12366.342} C_VEL
LIN {X 0,Y 385.085,Z 380.938,A -85,B 0,C 180,E1 -12368.904,E2 -12368.904} C_VEL
LIN {X 0,Y 383.844,Z 377.52,A -85,B 0,C 180,E1 -12371.35,E2 -12371.35} C_VEL
LIN {X 0,Y 383.39,Z 376.121,A -85,B 0,C 180,E1 -12372.841,E2 -12372.841} C_VEL
LIN {X 0,Y 383.004,Z 375.344,A -85,B 0,C 180,E1 -12374.305,E2 -12374.305} C_VEL
LIN {X 0,Y 382.815,Z 375.045,A -85,B 0,C 180,E1 -12375.763,E2 -12375.763} C_VEL
LIN {X 0,Y 382.866,Z 375.193,A -85,B 0,C 180,E1 -12377.244,E2 -12377.244} C_VEL
LIN {X 0,Y 383.123,Z 375.911,A -85,B 0,C 180,E1 -12378.773,E2 -12378.773} C_VEL
LIN {X 0,Y 383.544,Z 377.176,A -85,B 0,C 180,E1 -12380.318,E2 -12380.318} C_VEL
LIN {X 0,Y 384.645,Z 380.491,A -85,B 0,C 180,E1 -12382.918,E2 -12382.918} C_VEL
LIN {X 0,Y 385.808,Z 384.377,A -85,B 0,C 180,E1 -12385.059,E2 -12385.059} C_VEL
LIN {X 0,Y 387.285,Z 390.578,A -85,B 0,C 180,E1 -12387.673,E2 -12387.673} C_VEL
LIN {X 0,Y 388.514,Z 396.988,A -85,B 0,C 180,E1 -12389.886,E2 -12389.886} C_VEL
LIN {X 0,Y 388.928,Z 399.126,A -85,B 0,C 180,E1 -12390.493,E2 -12390.493} C_VEL
LIN {X 0,Y 391.063,Z 403.964,A -85,B 0,C 180,E1 -12391.132,E2 -12391.132} C_VEL
LIN {X 0,Y 394.079,Z 416.817,A -85,B 0,C 180,E1 -12392.202,E2 -12392.202} C_VEL
LIN {X 0,Y 396.615,Z 431.837,A -85,B 0,C 180,E1 -12393.215,E2 -12393.215} C_VEL
LIN {X 0,Y 396.453,Z 436.232,A -85,B 0,C 180,E1 -12393.377,E2 -12393.377} C_VEL
LIN {X 0,Y 390.745,Z 513.55,A -85,B 0,C 180,E1 -12395.741,E2 -12395.741} C_VEL
LIN {X 0,Y 388.589,Z 547.626,A -85,B 0,C 180,E1 -12396.801,E2 -12396.801} C_VEL
LIN {X 0,Y 387.322,Z 563.514,A -85,B 0,C 180,E1 -12397.531,E2 -12397.531} C_VEL
LIN {X 0,Y 385.927,Z 578.276,A -85,B 0,C 180,E1 -12398.457,E2 -12398.457} C_VEL
LIN {X 0,Y 384.395,Z 591.921,A -85,B 0,C 180,E1 -12399.533,E2 -12399.533} C_VEL
LIN {X 0,Y 382.783,Z 605.244,A -85,B 0,C 180,E1 -12400.841,E2 -12400.841} C_VEL
LIN {X 0,Y 381.306,Z 617.19,A -85,B 0,C 180,E1 -12402.295,E2 -12402.295} C_VEL
LIN {X 0,Y 379.843,Z 627.981,A -85,B 0,C 180,E1 -12403.887,E2 -12403.887} C_VEL
LIN {X 0,Y 378.537,Z 636.974,A -85,B 0,C 180,E1 -12405.485,E2 -12405.485} C_VEL
LIN {X 0,Y 377.362,Z 645.614,A -85,B 0,C 180,E1 -12407.36,E2 -12407.36} C_VEL
LIN {X 0,Y 376.473,Z 652.581,A -85,B 0,C 180,E1 -12409.241,E2 -12409.241} C_VEL
LIN {X 0,Y 375.908,Z 657.383,A -85,B 0,C 180,E1 -12410.856,E2 -12410.856} C_VEL
LIN {X 0,Y 375.33,Z 662.185,A -85,B 0,C 180,E1 -12412.942,E2 -12412.942} C_VEL
LIN {X 0,Y 374.955,Z 664.982,A -85,B 0,C 180,E1 -12414.623,E2 -12414.623} C_VEL
LIN {X 0,Y 374.897,Z 667.21,A -85,B 0,C 180,E1 -12416.776,E2 -12416.776} C_VEL
LIN {X 0,Y 374.65,Z 668.025,A -85,B 0,C 180,E1 -12418.925,E2 -12418.925} C_VEL
LIN {X 0,Y 374.638,Z 667.393,A -85,B 0,C 180,E1 -12421.075,E2 -12421.075} C_VEL
LIN {X 0,Y 374.689,Z 666.539,A -85,B 0,C 180,E1 -12422.15,E2 -12422.15} C_VEL
LIN {X 0,Y 374.701,Z 663.735,A -85,B 0,C 180,E1 -12424.303,E2 -12424.303} C_VEL
LIN {X 0,Y 374.893,Z 660.581,A -85,B 0,C 180,E1 -12425.918,E2 -12425.918} C_VEL
LIN {X 0,Y 375.082,Z 656.546,A -85,B 0,C 180,E1 -12427.537,E2 -12427.537} C_VEL
LIN {X 0,Y 375.352,Z 651.538,A -85,B 0,C 180,E1 -12429.158,E2 -12429.158} C_VEL
LIN {X 0,Y 375.898,Z 644.251,A -85,B 0,C 180,E1 -12431.049,E2 -12431.049} C_VEL
LIN {X 0,Y 376.692,Z 635.218,A -85,B 0,C 180,E1 -12432.937,E2 -12432.937} C_VEL
LIN {X 0,Y 377.465,Z 625.214,A -85,B 0,C 180,E1 -12434.651,E2 -12434.651} C_VEL
LIN {X 0,Y 378.366,Z 614.411,A -85,B 0,C 180,E1 -12436.178,E2 -12436.178} C_VEL
LIN {X 0,Y 379.346,Z 602.923,A -85,B 0,C 180,E1 -12437.521,E2 -12437.521} C_VEL
LIN {X 0,Y 380.443,Z 590.366,A -85,B 0,C 180,E1 -12438.722,E2 -12438.722} C_VEL
LIN {X 0,Y 381.381,Z 577.372,A -85,B 0,C 180,E1 -12439.731,E2 -12439.731} C_VEL
LIN {X 0,Y 382.32,Z 562.13,A -85,B 0,C 180,E1 -12440.654,E2 -12440.654} C_VEL
LIN {X 0,Y 383.078,Z 547.324,A -85,B 0,C 180,E1 -12441.314,E2 -12441.314} C_VEL
LIN {X 0,Y 383.651,Z 531.813,A -85,B 0,C 180,E1 -12441.775,E2 -12441.775} C_VEL
LIN {X 0,Y 386.866,Z 428.471,A -85,B 0,C 180,E1 -12444.278,E2 -12444.278} C_VEL
LIN {X 0,Y 381.75,Z 398.217,A -85,B 0,C 180,E1 -12445.379,E2 -12445.379} C_VEL
LIN {X 0,Y 382.009,Z 394.634,A -85,B 0,C 180,E1 -12445.984,E2 -12445.984} C_VEL
LIN {X 0,Y 382.724,Z 387.416,A -85,B 0,C 180,E1 -12447.328,E2 -12447.328} C_VEL
LIN {X 0,Y 379.96,Z 374.95,A -85,B 0,C 180,E1 -12449.961,E2 -12449.961} C_VEL
LIN {X 0,Y 376.093,Z 358.811,A -85,B 0,C 180,E1 -12453.533,E2 -12453.533} C_VEL
LIN {X 0,Y 376.013,Z 358.301,A -85,B 0,C 180,E1 -12453.783,E2 -12453.783} C_VEL
LIN {X 0,Y 375.948,Z 358.282,A -85,B 0,C 180,E1 -12456.742,E2 -12456.742} C_VEL
LIN {X 0,Y 375.939,Z 358.284,A -85,B 0,C 180,E1 -12459.961,E2 -12459.961} C_VEL
LIN {X 0,Y 375.925,Z 358.272,A -85,B 0,C 180,E1 -12463.767,E2 -12463.767} C_VEL
LIN {X 0,Y 375.933,Z 358.266,A -85,B 0,C 180,E1 -12466.811,E2 -12466.811} C_VEL
LIN {X 0,Y 375.933,Z 358.271,A -85,B 0,C 180,E1 -12470.533,E2 -12470.533} C_VEL
LIN {X 0,Y 375.973,Z 358.468,A -85,B 0,C 180,E1 -12473.031,E2 -12473.031} C_VEL
LIN {X 0,Y 379.659,Z 370.574,A -85,B 0,C 180,E1 -12475.462,E2 -12475.462} C_VEL
LIN {X 0,Y 383.097,Z 383.367,A -85,B 0,C 180,E1 -12477.858,E2 -12477.858} C_VEL
LIN {X 0,Y 385.605,Z 394.367,A -85,B 0,C 180,E1 -12479.763,E2 -12479.763} C_VEL
LIN {X 0,Y 385.588,Z 396.849,A -85,B 0,C 180,E1 -12480.1,E2 -12480.1} C_VEL
LIN {X 0,Y 390.617,Z 422.294,A -85,B 0,C 180,E1 -12481.057,E2 -12481.057} C_VEL
LIN {X 0,Y 392.623,Z 433.713,A -85,B 0,C 180,E1 -12481.452,E2 -12481.452} C_VEL
LIN {X 0,Y 389.611,Z 564.679,A -85,B 0,C 180,E1 -12483.916,E2 -12483.916} C_VEL
LIN {X 0,Y 388.786,Z 579.877,A -85,B 0,C 180,E1 -12484.386,E2 -12484.386} C_VEL
LIN {X 0,Y 387.724,Z 594.472,A -85,B 0,C 180,E1 -12485.043,E2 -12485.043} C_VEL
LIN {X 0,Y 386.534,Z 608.012,A -85,B 0,C 180,E1 -12485.852,E2 -12485.852} C_VEL
LIN {X 0,Y 385.007,Z 621.841,A -85,B 0,C 180,E1 -12486.892,E2 -12486.892} C_VEL
LIN {X 0,Y 383.485,Z 634.515,A -85,B 0,C 180,E1 -12488.074,E2 -12488.074} C_VEL
LIN {X 0,Y 381.9,Z 646.259,A -85,B 0,C 180,E1 -12489.393,E2 -12489.393} C_VEL
LIN {X 0,Y 380.439,Z 657.156,A -85,B 0,C 180,E1 -12490.858,E2 -12490.858} C_VEL
LIN {X 0,Y 379.364,Z 664.394,A -85,B 0,C 180,E1 -12491.992,E2 -12491.992} C_VEL
LIN {X 0,Y 378.187,Z 668.341,A -85,B 0,C 180,E1 -12492.638,E2 -12492.638} C_VEL
LIN {X 0,Y 374.55,Z 674.48,A -85,B 0,C 180,E1 -12493.683,E2 -12493.683} C_VEL
LIN {X 0,Y 370.938,Z 680.224,A -85,B 0,C 180,E1 -12494.797,E2 -12494.797} C_VEL
LIN {X 0,Y 369.82,Z 683.432,A -85,B 0,C 180,E1 -12495.543,E2 -12495.543} C_VEL
LIN {X 0,Y 369.036,Z 690.096,A -85,B 0,C 180,E1 -12497.349,E2 -12497.349} C_VEL
LIN {X 0,Y 368.212,Z 696.724,A -85,B 0,C 180,E1 -12499.553,E2 -12499.553} C_VEL
LIN {X 0,Y 367.759,Z 701.913,A -85,B 0,C 180,E1 -12501.759,E2 -12501.759} C_VEL
LIN {X 0,Y 367.45,Z 705.882,A -85,B 0,C 180,E1 -12504.029,E2 -12504.029} C_VEL
LIN {X 0,Y 367.405,Z 707.835,A -85,B 0,C 180,E1 -12505.612,E2 -12505.612} C_VEL
LIN {X 0,Y 367.312,Z 709.597,A -85,B 0,C 180,E1 -12507.807,E2 -12507.807} C_VEL
LIN {X 0,Y 367.341,Z 710.207,A -85,B 0,C 180,E1 -12510,E2 -12510} C_VEL
LIN {X 0,Y 367.313,Z 709.637,A -85,B 0,C 180,E1 -12512.193,E2 -12512.193} C_VEL
LIN {X 0,Y 367.41,Z 707.931,A -85,B 0,C 180,E1 -12514.388,E2 -12514.388} C_VEL
LIN {X 0,Y 367.556,Z 705.055,A -85,B 0,C 180,E1 -12516.588,E2 -12516.588} C_VEL
LIN {X 0,Y 367.846,Z 700.941,A -85,B 0,C 180,E1 -12518.792,E2 -12518.792} C_VEL
LIN {X 0,Y 368.325,Z 695.48,A -85,B 0,C 180,E1 -12521,E2 -12521} C_VEL
LIN {X 0,Y 369.191,Z 688.523,A -85,B 0,C 180,E1 -12523.205,E2 -12523.205} C_VEL
LIN {X 0,Y 370.165,Z 681.078,A -85,B 0,C 180,E1 -12525.133,E2 -12525.133} C_VEL
LIN {X 0,Y 371.46,Z 672.108,A -85,B 0,C 180,E1 -12527.053,E2 -12527.053} C_VEL
LIN {X 0,Y 373.141,Z 661.267,A -85,B 0,C 180,E1 -12528.959,E2 -12528.959} C_VEL
LIN {X 0,Y 374.65,Z 650.243,A -85,B 0,C 180,E1 -12530.578,E2 -12530.578} C_VEL
LIN {X 0,Y 376.442,Z 637.92,A -85,B 0,C 180,E1 -12532.069,E2 -12532.069} C_VEL
LIN {X 0,Y 378.188,Z 624.438,A -85,B 0,C 180,E1 -12533.404,E2 -12533.404} C_VEL
LIN {X 0,Y 379.733,Z 611.251,A -85,B 0,C 180,E1 -12534.463,E2 -12534.463} C_VEL
LIN {X 0,Y 381.086,Z 597.305,A -85,B 0,C 180,E1 -12535.356,E2 -12535.356} C_VEL
LIN {X 0,Y 382.18,Z 583.283,A -85,B 0,C 180,E1 -12536.043,E2 -12536.043} C_VEL
LIN {X 0,Y 383.128,Z 568.247,A -85,B 0,C 180,E1 -12536.559,E2 -12536.559} C_VEL
LIN {X 0,Y 383.774,Z 546.183,A -85,B 0,C 180,E1 -12537.025,E2 -12537.025} C_VEL
LIN {X 0,Y 386.375,Z 434.341,A -85,B 0,C 180,E1 -12539.141,E2 -12539.141} C_VEL
LIN {X 0,Y 381.431,Z 407.762,A -85,B 0,C 180,E1 -12540.12,E2 -12540.12} C_VEL
LIN {X 0,Y 379.059,Z 396.368,A -85,B 0,C 180,E1 -12540.61,E2 -12540.61} C_VEL
LIN {X 0,Y 375.592,Z 381.892,A -85,B 0,C 180,E1 -12543.183,E2 -12543.183} C_VEL
LIN {X 0,Y 371.616,Z 367.86,A -85,B 0,C 180,E1 -12545.893,E2 -12545.893} C_VEL
LIN {X 0,Y 368.932,Z 359.336,A -85,B 0,C 180,E1 -12547.689,E2 -12547.689} C_VEL
LIN {X 0,Y 368.883,Z 359.147,A -85,B 0,C 180,E1 -12550.374,E2 -12550.374} C_VEL
LIN {X 0,Y 368.881,Z 359.162,A -85,B 0,C 180,E1 -12553.615,E2 -12553.615} C_VEL
LIN {X 0,Y 368.885,Z 359.162,A -85,B 0,C 180,E1 -12556.696,E2 -12556.696} C_VEL
LIN {X 0,Y 368.884,Z 359.164,A -85,B 0,C 180,E1 -12559.648,E2 -12559.648} C_VEL
LIN {X 0,Y 368.895,Z 359.16,A -85,B 0,C 180,E1 -12563.145,E2 -12563.145} C_VEL
LIN {X 0,Y 368.895,Z 359.158,A -85,B 0,C 180,E1 -12566.462,E2 -12566.462} C_VEL
LIN {X 0,Y 368.913,Z 359.146,A -85,B 0,C 180,E1 -12569.045,E2 -12569.045} C_VEL
LIN {X 0,Y 368.916,Z 359.152,A -85,B 0,C 180,E1 -12571.558,E2 -12571.558} C_VEL
LIN {X 0,Y 368.914,Z 359.156,A -85,B 0,C 180,E1 -12575.221,E2 -12575.221} C_VEL
LIN {X 0,Y 368.91,Z 359.147,A -85,B 0,C 180,E1 -12578.779,E2 -12578.779} C_VEL
LIN {X 0,Y 368.991,Z 359.135,A -85,B 0,C 180,E1 -12582.257,E2 -12582.257} C_VEL
LIN {X 0,Y 369.038,Z 359.14,A -85,B 0,C 180,E1 -12586.228,E2 -12586.228} C_VEL
LIN {X 0,Y 369.064,Z 359.127,A -85,B 0,C 180,E1 -12590.132,E2 -12590.132} C_VEL
LIN {X 0,Y 369.189,Z 359.115,A -85,B 0,C 180,E1 -12593.441,E2 -12593.441} C_VEL
LIN {X 0,Y 369.308,Z 359.108,A -85,B 0,C 180,E1 -12597.819,E2 -12597.819} C_VEL
LIN {X 0,Y 369.455,Z 359.079,A -85,B 0,C 180,E1 -12600,E2 -12600} C_VEL
LIN {X 0,Y 369.315,Z 359.09,A -85,B 0,C 180,E1 -12602.181,E2 -12602.181} C_VEL
LIN {X 0,Y 369.174,Z 359.114,A -85,B 0,C 180,E1 -12606.559,E2 -12606.559} C_VEL
LIN {X 0,Y 369.064,Z 359.135,A -85,B 0,C 180,E1 -12609.868,E2 -12609.868} C_VEL
LIN {X 0,Y 369.037,Z 359.121,A -85,B 0,C 180,E1 -12613.772,E2 -12613.772} C_VEL
LIN {X 0,Y 368.991,Z 359.141,A -85,B 0,C 180,E1 -12617.743,E2 -12617.743} C_VEL
LIN {X 0,Y 368.93,Z 359.148,A -85,B 0,C 180,E1 -12621.219,E2 -12621.219} C_VEL
LIN {X 0,Y 368.958,Z 359.137,A -85,B 0,C 180,E1 -12624.775,E2 -12624.775} C_VEL
LIN {X 0,Y 368.968,Z 359.152,A -85,B 0,C 180,E1 -12627.203,E2 -12627.203} C_VEL
LIN {X 0,Y 368.919,Z 359.142,A -85,B 0,C 180,E1 -12629.69,E2 -12629.69} C_VEL
LIN {X 0,Y 368.897,Z 359.156,A -85,B 0,C 180,E1 -12633.043,E2 -12633.043} C_VEL
LIN {X 0,Y 368.917,Z 359.155,A -85,B 0,C 180,E1 -12636.197,E2 -12636.197} C_VEL
LIN {X 0,Y 368.9,Z 359.126,A -85,B 0,C 180,E1 -12638.953,E2 -12638.953} C_VEL
LIN {X 0,Y 368.881,Z 359.138,A -85,B 0,C 180,E1 -12642.009,E2 -12642.009} C_VEL
LIN {X 0,Y 368.88,Z 359.146,A -85,B 0,C 180,E1 -12645.176,E2 -12645.176} C_VEL
LIN {X 0,Y 368.882,Z 359.142,A -85,B 0,C 180,E1 -12648.178,E2 -12648.178} C_VEL
LIN {X 0,Y 368.908,Z 359.159,A -85,B 0,C 180,E1 -12651.36,E2 -12651.36} C_VEL
LIN {X 0,Y 368.97,Z 359.369,A -85,B 0,C 180,E1 -12653.497,E2 -12653.497} C_VEL
LIN {X 0,Y 373.078,Z 374.792,A -85,B 0,C 180,E1 -12656.645,E2 -12656.645} C_VEL
LIN {X 0,Y 376.691,Z 388.481,A -85,B 0,C 180,E1 -12659.249,E2 -12659.249} C_VEL
LIN {X 0,Y 377.986,Z 392.126,A -85,B 0,C 180,E1 -12659.557,E2 -12659.557} C_VEL
LIN {X 0,Y 380.146,Z 397.582,A -85,B 0,C 180,E1 -12659.866,E2 -12659.866} C_VEL
LIN {X 0,Y 385.783,Z 432.175,A -85,B 0,C 180,E1 -12661.076,E2 -12661.076} C_VEL
LIN {X 0,Y 382.681,Z 564.476,A -85,B 0,C 180,E1 -12663.591,E2 -12663.591} C_VEL
LIN {X 0,Y 381.811,Z 579.976,A -85,B 0,C 180,E1 -12664.077,E2 -12664.077} C_VEL
LIN {X 0,Y 380.661,Z 595.104,A -85,B 0,C 180,E1 -12664.778,E2 -12664.778} C_VEL
LIN {X 0,Y 379.387,Z 609.748,A -85,B 0,C 180,E1 -12665.699,E2 -12665.699} C_VEL
LIN {X 0,Y 377.652,Z 624.214,A -85,B 0,C 180,E1 -12666.851,E2 -12666.851} C_VEL
LIN {X 0,Y 375.947,Z 637.582,A -85,B 0,C 180,E1 -12668.189,E2 -12668.189} C_VEL
LIN {X 0,Y 374.303,Z 649.72,A -85,B 0,C 180,E1 -12669.675,E2 -12669.675} C_VEL
LIN {X 0,Y 372.751,Z 660.774,A -85,B 0,C 180,E1 -12671.305,E2 -12671.305} C_VEL
LIN {X 0,Y 371.352,Z 670.078,A -85,B 0,C 180,E1 -12672.942,E2 -12672.942} C_VEL
LIN {X 0,Y 370.067,Z 679.199,A -85,B 0,C 180,E1 -12674.863,E2 -12674.863} C_VEL
LIN {X 0,Y 369.09,Z 686.762,A -85,B 0,C 180,E1 -12676.792,E2 -12676.792} C_VEL
LIN {X 0,Y 368.287,Z 693.816,A -85,B 0,C 180,E1 -12678.999,E2 -12678.999} C_VEL
LIN {X 0,Y 367.836,Z 699.354,A -85,B 0,C 180,E1 -12681.208,E2 -12681.208} C_VEL
LIN {X 0,Y 367.552,Z 703.528,A -85,B 0,C 180,E1 -12683.412,E2 -12683.412} C_VEL
LIN {X 0,Y 367.41,Z 706.451,A -85,B 0,C 180,E1 -12685.612,E2 -12685.612} C_VEL
LIN {X 0,Y 367.359,Z 708.196,A -85,B 0,C 180,E1 -12687.807,E2 -12687.807} C_VEL
LIN {X 0,Y 367.34,Z 708.791,A -85,B 0,C 180,E1 -12690,E2 -12690} C_VEL
LIN {X 0,Y 367.362,Z 708.194,A -85,B 0,C 180,E1 -12692.193,E2 -12692.193} C_VEL
LIN {X 0,Y 367.41,Z 706.447,A -85,B 0,C 180,E1 -12694.388,E2 -12694.388} C_VEL
LIN {X 0,Y 367.552,Z 703.514,A -85,B 0,C 180,E1 -12696.588,E2 -12696.588} C_VEL
LIN {X 0,Y 367.837,Z 699.328,A -85,B 0,C 180,E1 -12698.792,E2 -12698.792} C_VEL
LIN {X 0,Y 368.29,Z 693.787,A -85,B 0,C 180,E1 -12701.001,E2 -12701.001} C_VEL
LIN {X 0,Y 368.932,Z 688.66,A -85,B 0,C 180,E1 -12702.655,E2 -12702.655} C_VEL
LIN {X 0,Y 369.953,Z 680.343,A -85,B 0,C 180,E1 -12704.86,E2 -12704.86} C_VEL
LIN {X 0,Y 371.176,Z 671.433,A -85,B 0,C 180,E1 -12706.783,E2 -12706.783} C_VEL
LIN {X 0,Y 372.453,Z 662.331,A -85,B 0,C 180,E1 -12708.425,E2 -12708.425} C_VEL
LIN {X 0,Y 373.948,Z 651.987,A -85,B 0,C 180,E1 -12709.999,E2 -12709.999} C_VEL
LIN {X 0,Y 375.626,Z 639.81,A -85,B 0,C 180,E1 -12711.542,E2 -12711.542} C_VEL
LIN {X 0,Y 377.325,Z 626.931,A -85,B 0,C 180,E1 -12712.881,E2 -12712.881} C_VEL
LIN {X 0,Y 378.799,Z 614.422,A -85,B 0,C 180,E1 -12713.945,E2 -12713.945} C_VEL
LIN {X 0,Y 380.198,Z 600.593,A -85,B 0,C 180,E1 -12714.889,E2 -12714.889} C_VEL
LIN {X 0,Y 381.435,Z 585.835,A -85,B 0,C 180,E1 -12715.66,E2 -12715.66} C_VEL
LIN {X 0,Y 383.406,Z 559.182,A -85,B 0,C 180,E1 -12716.686,E2 -12716.686} C_VEL
LIN {X 0,Y 388.567,Z 476.721,A -85,B 0,C 180,E1 -12718.973,E2 -12718.973} C_VEL
LIN {X 0,Y 391.735,Z 432.158,A -85,B 0,C 180,E1 -12720.301,E2 -12720.301} C_VEL
LIN {X 0,Y 390.237,Z 418.819,A -85,B 0,C 180,E1 -12721.088,E2 -12721.088} C_VEL
LIN {X 0,Y 388.613,Z 409.637,A -85,B 0,C 180,E1 -12721.752,E2 -12721.752} C_VEL
LIN {X 0,Y 385.12,Z 402.748,A -85,B 0,C 180,E1 -12722.688,E2 -12722.688} C_VEL
LIN {X 0,Y 383.172,Z 398.898,A -85,B 0,C 180,E1 -12723.311,E2 -12723.311} C_VEL
LIN {X 0,Y 381.769,Z 393.039,A -85,B 0,C 180,E1 -12725.339,E2 -12725.339} C_VEL
LIN {X 0,Y 380.271,Z 387.87,A -85,B 0,C 180,E1 -12727.582,E2 -12727.582} C_VEL
LIN {X 0,Y 379.463,Z 385.181,A -85,B 0,C 180,E1 -12729.029,E2 -12729.029} C_VEL
LIN {X 0,Y 378.677,Z 383.043,A -85,B 0,C 180,E1 -12730.51,E2 -12730.51} C_VEL
LIN {X 0,Y 378.096,Z 381.364,A -85,B 0,C 180,E1 -12732.003,E2 -12732.003} C_VEL
LIN {X 0,Y 377.677,Z 380.191,A -85,B 0,C 180,E1 -12733.513,E2 -12733.513} C_VEL
LIN {X 0,Y 377.36,Z 379.633,A -85,B 0,C 180,E1 -12735.05,E2 -12735.05} C_VEL
LIN {X 0,Y 377.297,Z 379.584,A -85,B 0,C 180,E1 -12736.591,E2 -12736.591} C_VEL
LIN {X 0,Y 377.443,Z 380.045,A -85,B 0,C 180,E1 -12738.142,E2 -12738.142} C_VEL
LIN {X 0,Y 377.784,Z 381.033,A -85,B 0,C 180,E1 -12739.706,E2 -12739.706} C_VEL
LIN {X 0,Y 378.657,Z 383.833,A -85,B 0,C 180,E1 -12742.23,E2 -12742.23} C_VEL
LIN {X 0,Y 379.755,Z 387.583,A -85,B 0,C 180,E1 -12744.518,E2 -12744.518} C_VEL
LIN {X 0,Y 380.738,Z 391.469,A -85,B 0,C 180,E1 -12746.374,E2 -12746.374} C_VEL
LIN {X 0,Y 382.089,Z 398.291,A -85,B 0,C 180,E1 -12749.001,E2 -12749.001} C_VEL
LIN {X 0,Y 382.435,Z 399.588,A -85,B 0,C 180,E1 -12749.323,E2 -12749.323} C_VEL
LIN {X 0,Y 386.485,Z 407.534,A -85,B 0,C 180,E1 -12750.533,E2 -12750.533} C_VEL
LIN {X 0,Y 389.237,Z 420.248,A -85,B 0,C 180,E1 -12751.624,E2 -12751.624} C_VEL
LIN {X 0,Y 391.425,Z 434.144,A -85,B 0,C 180,E1 -12752.6,E2 -12752.6} C_VEL
LIN {X 0,Y 385.266,Z 510.486,A -85,B 0,C 180,E1 -12755.013,E2 -12755.013} C_VEL
LIN {X 0,Y 382.724,Z 547.681,A -85,B 0,C 180,E1 -12756.208,E2 -12756.208} C_VEL
LIN {X 0,Y 381.352,Z 563.436,A -85,B 0,C 180,E1 -12756.945,E2 -12756.945} C_VEL
LIN {X 0,Y 379.908,Z 577.882,A -85,B 0,C 180,E1 -12757.859,E2 -12757.859} C_VEL
LIN {X 0,Y 378.148,Z 592.549,A -85,B 0,C 180,E1 -12759.037,E2 -12759.037} C_VEL
LIN {X 0,Y 376.41,Z 605.763,A -85,B 0,C 180,E1 -12760.362,E2 -12760.362} C_VEL
LIN {X 0,Y 374.966,Z 616.677,A -85,B 0,C 180,E1 -12761.703,E2 -12761.703} C_VEL
LIN {X 0,Y 373.401,Z 627.579,A -85,B 0,C 180,E1 -12763.32,E2 -12763.32} C_VEL
LIN {X 0,Y 371.99,Z 636.682,A -85,B 0,C 180,E1 -12764.943,E2 -12764.943} C_VEL
LIN {X 0,Y 370.668,Z 645.429,A -85,B 0,C 180,E1 -12766.849,E2 -12766.849} C_VEL
LIN {X 0,Y 369.776,Z 651.586,A -85,B 0,C 180,E1 -12768.489,E2 -12768.489} C_VEL
LIN {X 0,Y 369.164,Z 656.676,A -85,B 0,C 180,E1 -12770.134,E2 -12770.134} C_VEL
LIN {X 0,Y 368.432,Z 661.892,A -85,B 0,C 180,E1 -12772.327,E2 -12772.327} C_VEL
LIN {X 0,Y 368.214,Z 663.899,A -85,B 0,C 180,E1 -12773.424,E2 -12773.424} C_VEL
LIN {X 0,Y 367.817,Z 666.791,A -85,B 0,C 180,E1 -12775.617,E2 -12775.617} C_VEL
LIN {X 0,Y 367.823,Z 667.684,A -85,B 0,C 180,E1 -12776.714,E2 -12776.714} C_VEL
LIN {X 0,Y 367.586,Z 668.413,A -85,B 0,C 180,E1 -12778.905,E2 -12778.905} C_VEL
LIN {X 0,Y 367.574,Z 667.694,A -85,B 0,C 180,E1 -12781.096,E2 -12781.096} C_VEL
LIN {X 0,Y 367.593,Z 666.796,A -85,B 0,C 180,E1 -12782.192,E2 -12782.192} C_VEL
LIN {X 0,Y 367.633,Z 663.875,A -85,B 0,C 180,E1 -12784.386,E2 -12784.386} C_VEL
LIN {X 0,Y 367.823,Z 660.353,A -85,B 0,C 180,E1 -12786.172,E2 -12786.172} C_VEL
LIN {X 0,Y 368.084,Z 654.955,A -85,B 0,C 180,E1 -12788.233,E2 -12788.233} C_VEL
LIN {X 0,Y 368.577,Z 648.442,A -85,B 0,C 180,E1 -12790.159,E2 -12790.159} C_VEL
LIN {X 0,Y 369.177,Z 640.298,A -85,B 0,C 180,E1 -12792.088,E2 -12792.088} C_VEL
LIN {X 0,Y 369.941,Z 631.822,A -85,B 0,C 180,E1 -12793.737,E2 -12793.737} C_VEL
LIN {X 0,Y 370.775,Z 621.606,A -85,B 0,C 180,E1 -12795.389,E2 -12795.389} C_VEL
LIN {X 0,Y 371.787,Z 610.323,A -85,B 0,C 180,E1 -12796.896,E2 -12796.896} C_VEL
LIN {X 0,Y 372.848,Z 597.917,A -85,B 0,C 180,E1 -12798.263,E2 -12798.263} C_VEL
LIN {X 0,Y 373.872,Z 585.844,A -85,B 0,C 180,E1 -12799.349,E2 -12799.349} C_VEL
LIN {X 0,Y 374.877,Z 571.435,A -85,B 0,C 180,E1 -12800.384,E2 -12800.384} C_VEL
LIN {X 0,Y 375.696,Z 557.056,A -85,B 0,C 180,E1 -12801.178,E2 -12801.178} C_VEL
LIN {X 0,Y 376.492,Z 541.969,A -85,B 0,C 180,E1 -12801.778,E2 -12801.778} C_VEL
LIN {X 0,Y 380.121,Z 429.218,A -85,B 0,C 180,E1 -12804.626,E2 -12804.626} C_VEL
LIN {X 0,Y 374.976,Z 397.801,A -85,B 0,C 180,E1 -12805.806,E2 -12805.806} C_VEL
LIN {X 0,Y 375.757,Z 388.446,A -85,B 0,C 180,E1 -12807.575,E2 -12807.575} C_VEL
LIN {X 0,Y 372.542,Z 374.318,A -85,B 0,C 180,E1 -12810.621,E2 -12810.621} C_VEL
LIN {X 0,Y 368.978,Z 359.401,A -85,B 0,C 180,E1 -12814.022,E2 -12814.022} C_VEL
LIN {X 0,Y 368.923,Z 359.157,A -85,B 0,C 180,E1 -12815,E2 -12815} C_VEL
LIN {X 0,Y 368.876,Z 359.162,A -85,B 0,C 180,E1 -12818.634,E2 -12818.634} C_VEL
LIN {X 0,Y 368.858,Z 359.146,A -85,B 0,C 180,E1 -12822.005,E2 -12822.005} C_VEL
LIN {X 0,Y 368.874,Z 359.163,A -85,B 0,C 180,E1 -12825.175,E2 -12825.175} C_VEL
LIN {X 0,Y 368.86,Z 359.157,A -85,B 0,C 180,E1 -12828.174,E2 -12828.174} C_VEL
LIN {X 0,Y 368.892,Z 359.159,A -85,B 0,C 180,E1 -12831.744,E2 -12831.744} C_VEL
LIN {X 0,Y 368.941,Z 359.458,A -85,B 0,C 180,E1 -12832.466,E2 -12832.466} C_VEL
LIN {X 0,Y 372.853,Z 372.066,A -85,B 0,C 180,E1 -12835.046,E2 -12835.046} C_VEL
LIN {X 0,Y 376.519,Z 385.609,A -85,B 0,C 180,E1 -12837.615,E2 -12837.615} C_VEL
LIN {X 0,Y 379.065,Z 396.562,A -85,B 0,C 180,E1 -12839.518,E2 -12839.518} C_VEL
LIN {X 0,Y 383.912,Z 420.739,A -85,B 0,C 180,E1 -12840.472,E2 -12840.472} C_VEL
LIN {X 0,Y 386.341,Z 434.005,A -85,B 0,C 180,E1 -12840.952,E2 -12840.952} C_VEL
LIN {X 0,Y 383.706,Z 548.338,A -85,B 0,C 180,E1 -12843.116,E2 -12843.116} C_VEL
LIN {X 0,Y 383.074,Z 568.458,A -85,B 0,C 180,E1 -12843.546,E2 -12843.546} C_VEL
LIN {X 0,Y 382.081,Z 583.856,A -85,B 0,C 180,E1 -12844.082,E2 -12844.082} C_VEL
LIN {X 0,Y 380.946,Z 598.817,A -85,B 0,C 180,E1 -12844.835,E2 -12844.835} C_VEL
LIN {X 0,Y 379.69,Z 611.825,A -85,B 0,C 180,E1 -12845.679,E2 -12845.679} C_VEL
LIN {X 0,Y 378.11,Z 624.898,A -85,B 0,C 180,E1 -12846.735,E2 -12846.735} C_VEL
LIN {X 0,Y 376.346,Z 638.283,A -85,B 0,C 180,E1 -12848.069,E2 -12848.069} C_VEL
LIN {X 0,Y 374.54,Z 650.969,A -85,B 0,C 180,E1 -12849.619,E2 -12849.619} C_VEL
LIN {X 0,Y 372.936,Z 662.374,A -85,B 0,C 180,E1 -12851.315,E2 -12851.315} C_VEL
LIN {X 0,Y 371.324,Z 672.991,A -85,B 0,C 180,E1 -12853.224,E2 -12853.224} C_VEL
LIN {X 0,Y 370.053,Z 681.83,A -85,B 0,C 180,E1 -12855.144,E2 -12855.144} C_VEL
LIN {X 0,Y 369.82,Z 683.432,A -85,B 0,C 180,E1 -12855.543,E2 -12855.543} C_VEL
LIN {X 0,Y 368.733,Z 686.52,A -85,B 0,C 180,E1 -12856.311,E2 -12856.311} C_VEL
LIN {X 0,Y 365.29,Z 691.195,A -85,B 0,C 180,E1 -12857.567,E2 -12857.567} C_VEL
LIN {X 0,Y 361.968,Z 695.416,A -85,B 0,C 180,E1 -12858.885,E2 -12858.885} C_VEL
LIN {X 0,Y 361.088,Z 697.686,A -85,B 0,C 180,E1 -12859.738,E2 -12859.738} C_VEL
LIN {X 0,Y 360.594,Z 702.954,A -85,B 0,C 180,E1 -12862.158,E2 -12862.158} C_VEL
LIN {X 0,Y 360.338,Z 706.504,A -85,B 0,C 180,E1 -12864.403,E2 -12864.403} C_VEL
LIN {X 0,Y 360.261,Z 708.846,A -85,B 0,C 180,E1 -12866.645,E2 -12866.645} C_VEL
LIN {X 0,Y 360.245,Z 710.037,A -85,B 0,C 180,E1 -12868.882,E2 -12868.882} C_VEL
LIN {X 0,Y 360.246,Z 710.05,A -85,B 0,C 180,E1 -12871.118,E2 -12871.118} C_VEL
LIN {X 0,Y 360.262,Z 708.913,A -85,B 0,C 180,E1 -12873.355,E2 -12873.355} C_VEL
LIN {X 0,Y 360.359,Z 706.628,A -85,B 0,C 180,E1 -12875.596,E2 -12875.596} C_VEL
LIN {X 0,Y 360.627,Z 703.143,A -85,B 0,C 180,E1 -12877.84,E2 -12877.84} C_VEL
LIN {X 0,Y 361.033,Z 698.371,A -85,B 0,C 180,E1 -12880.09,E2 -12880.09} C_VEL
LIN {X 0,Y 361.797,Z 692.182,A -85,B 0,C 180,E1 -12882.338,E2 -12882.338} C_VEL
LIN {X 0,Y 362.759,Z 684.404,A -85,B 0,C 180,E1 -12884.587,E2 -12884.587} C_VEL
LIN {X 0,Y 364.006,Z 676.115,A -85,B 0,C 180,E1 -12886.546,E2 -12886.546} C_VEL
LIN {X 0,Y 365.527,Z 666.125,A -85,B 0,C 180,E1 -12888.496,E2 -12888.496} C_VEL
LIN {X 0,Y 367.114,Z 655.926,A -85,B 0,C 180,E1 -12890.157,E2 -12890.157} C_VEL
LIN {X 0,Y 368.95,Z 643.712,A -85,B 0,C 180,E1 -12891.805,E2 -12891.805} C_VEL
LIN {X 0,Y 370.708,Z 631.495,A -85,B 0,C 180,E1 -12893.165,E2 -12893.165} C_VEL
LIN {X 0,Y 372.43,Z 618.156,A -85,B 0,C 180,E1 -12894.38,E2 -12894.38} C_VEL
LIN {X 0,Y 373.975,Z 604.342,A -85,B 0,C 180,E1 -12895.391,E2 -12895.391} C_VEL
LIN {X 0,Y 375.292,Z 589.032,A -85,B 0,C 180,E1 -12896.258,E2 -12896.258} C_VEL
LIN {X 0,Y 376.406,Z 574.513,A -85,B 0,C 180,E1 -12896.847,E2 -12896.847} C_VEL
LIN {X 0,Y 377.164,Z 558.42,A -85,B 0,C 180,E1 -12897.276,E2 -12897.276} C_VEL
LIN {X 0,Y 380.164,Z 435.401,A -85,B 0,C 180,E1 -12899.638,E2 -12899.638} C_VEL
LIN {X 0,Y 375.441,Z 409.907,A -85,B 0,C 180,E1 -12900.601,E2 -12900.601} C_VEL
LIN {X 0,Y 373.019,Z 398.899,A -85,B 0,C 180,E1 -12901.062,E2 -12901.062} C_VEL
LIN {X 0,Y 371.962,Z 396.255,A -85,B 0,C 180,E1 -12901.261,E2 -12901.261} C_VEL
LIN {X 0,Y 368.64,Z 382.654,A -85,B 0,C 180,E1 -12903.737,E2 -12903.737} C_VEL
LIN {X 0,Y 365.229,Z 370.734,A -85,B 0,C 180,E1 -12906.08,E2 -12906.08} C_VEL
LIN {X 0,Y 361.872,Z 360.239,A -85,B 0,C 180,E1 -12908.317,E2 -12908.317} C_VEL
LIN {X 0,Y 361.811,Z 360.042,A -85,B 0,C 180,E1 -12911.333,E2 -12911.333} C_VEL
LIN {X 0,Y 361.814,Z 360.039,A -85,B 0,C 180,E1 -12914.369,E2 -12914.369} C_VEL
LIN {X 0,Y 361.829,Z 360.036,A -85,B 0,C 180,E1 -12917.569,E2 -12917.569} C_VEL
LIN {X 0,Y 361.842,Z 360.032,A -85,B 0,C 180,E1 -12921.572,E2 -12921.572} C_VEL
LIN {X 0,Y 361.87,Z 360.024,A -85,B 0,C 180,E1 -12924.656,E2 -12924.656} C_VEL
LIN {X 0,Y 361.837,Z 360.025,A -85,B 0,C 180,E1 -12928.37,E2 -12928.37} C_VEL
LIN {X 0,Y 361.866,Z 360.034,A -85,B 0,C 180,E1 -12930.952,E2 -12930.952} C_VEL
LIN {X 0,Y 361.876,Z 360.031,A -85,B 0,C 180,E1 -12934.706,E2 -12934.706} C_VEL
LIN {X 0,Y 361.854,Z 360.022,A -85,B 0,C 180,E1 -12938.345,E2 -12938.345} C_VEL
LIN {X 0,Y 361.92,Z 360.016,A -85,B 0,C 180,E1 -12942.085,E2 -12942.085} C_VEL
LIN {X 0,Y 361.962,Z 360.02,A -85,B 0,C 180,E1 -12945.38,E2 -12945.38} C_VEL
LIN {X 0,Y 361.971,Z 360.003,A -85,B 0,C 180,E1 -12948.804,E2 -12948.804} C_VEL
LIN {X 0,Y 362.096,Z 360.004,A -85,B 0,C 180,E1 -12952.191,E2 -12952.191} C_VEL
LIN {X 0,Y 362.111,Z 359.988,A -85,B 0,C 180,E1 -12954.431,E2 -12954.431} C_VEL
LIN {X 0,Y 362.271,Z 359.985,A -85,B 0,C 180,E1 -12957.776,E2 -12957.776} C_VEL
LIN {X 0,Y 362.425,Z 359.954,A -85,B 0,C 180,E1 -12960,E2 -12960} C_VEL
LIN {X 0,Y 362.279,Z 359.966,A -85,B 0,C 180,E1 -12962.223,E2 -12962.223} C_VEL
LIN {X 0,Y 362.136,Z 359.988,A -85,B 0,C 180,E1 -12966.687,E2 -12966.687} C_VEL
LIN {X 0,Y 362.001,Z 360.014,A -85,B 0,C 180,E1 -12970.063,E2 -12970.063} C_VEL
LIN {X 0,Y 361.998,Z 359.997,A -85,B 0,C 180,E1 -12973.899,E2 -12973.899} C_VEL
LIN {X 0,Y 361.928,Z 360.027,A -85,B 0,C 180,E1 -12976.934,E2 -12976.934} C_VEL
LIN {X 0,Y 361.894,Z 360.018,A -85,B 0,C 180,E1 -12980.46,E2 -12980.46} C_VEL
LIN {X 0,Y 361.895,Z 360.021,A -85,B 0,C 180,E1 -12984.114,E2 -12984.114} C_VEL
LIN {X 0,Y 361.942,Z 360.021,A -85,B 0,C 180,E1 -12986.722,E2 -12986.722} C_VEL
LIN {X 0,Y 361.874,Z 360.02,A -85,B 0,C 180,E1 -12990.328,E2 -12990.328} C_VEL
LIN {X 0,Y 361.854,Z 360.024,A -85,B 0,C 180,E1 -12994.28,E2 -12994.28} C_VEL
LIN {X 0,Y 361.863,Z 360.031,A -85,B 0,C 180,E1 -12997.223,E2 -12997.223} C_VEL
LIN {X 0,Y 361.834,Z 359.995,A -85,B 0,C 180,E1 -13000.755,E2 -13000.755} C_VEL
LIN {X 0,Y 361.819,Z 360.038,A -85,B 0,C 180,E1 -13004.368,E2 -13004.368} C_VEL
LIN {X 0,Y 361.835,Z 360.009,A -85,B 0,C 180,E1 -13007.568,E2 -13007.568} C_VEL
LIN {X 0,Y 361.87,Z 360.036,A -85,B 0,C 180,E1 -13010.973,E2 -13010.973} C_VEL
LIN {X 0,Y 361.882,Z 360.192,A -85,B 0,C 180,E1 -13013.017,E2 -13013.017} C_VEL
LIN {X 0,Y 365.862,Z 375.09,A -85,B 0,C 180,E1 -13016.146,E2 -13016.146} C_VEL
LIN {X 0,Y 368.91,Z 386.606,A -85,B 0,C 180,E1 -13018.39,E2 -13018.39} C_VEL
LIN {X 0,Y 370.89,Z 391.887,A -85,B 0,C 180,E1 -13018.901,E2 -13018.901} C_VEL
LIN {X 0,Y 374.168,Z 399.564,A -85,B 0,C 180,E1 -13019.373,E2 -13019.373} C_VEL
LIN {X 0,Y 379.556,Z 432.751,A -85,B 0,C 180,E1 -13020.564,E2 -13020.564} C_VEL
LIN {X 0,Y 376.339,Z 564.596,A -85,B 0,C 180,E1 -13023.11,E2 -13023.11} C_VEL
LIN {X 0,Y 375.457,Z 579.773,A -85,B 0,C 180,E1 -13023.593,E2 -13023.593} C_VEL
LIN {X 0,Y 374.249,Z 594.938,A -85,B 0,C 180,E1 -13024.302,E2 -13024.302} C_VEL
LIN {X 0,Y 372.898,Z 609.975,A -85,B 0,C 180,E1 -13025.263,E2 -13025.263} C_VEL
LIN {X 0,Y 371.105,Z 624.247,A -85,B 0,C 180,E1 -13026.418,E2 -13026.418} C_VEL
LIN {X 0,Y 369.355,Z 637.61,A -85,B 0,C 180,E1 -13027.779,E2 -13027.779} C_VEL
LIN {X 0,Y 367.589,Z 649.745,A -85,B 0,C 180,E1 -13029.287,E2 -13029.287} C_VEL
LIN {X 0,Y 365.987,Z 660.796,A -85,B 0,C 180,E1 -13030.947,E2 -13030.947} C_VEL
LIN {X 0,Y 364.525,Z 670.099,A -85,B 0,C 180,E1 -13032.612,E2 -13032.612} C_VEL
LIN {X 0,Y 363.159,Z 679.218,A -85,B 0,C 180,E1 -13034.568,E2 -13034.568} C_VEL
LIN {X 0,Y 362.139,Z 686.779,A -85,B 0,C 180,E1 -13036.533,E2 -13036.533} C_VEL
LIN {X 0,Y 361.269,Z 693.832,A -85,B 0,C 180,E1 -13038.782,E2 -13038.782} C_VEL
LIN {X 0,Y 360.78,Z 699.369,A -85,B 0,C 180,E1 -13041.035,E2 -13041.035} C_VEL
LIN {X 0,Y 360.483,Z 703.543,A -85,B 0,C 180,E1 -13043.282,E2 -13043.282} C_VEL
LIN {X 0,Y 360.323,Z 706.466,A -85,B 0,C 180,E1 -13045.525,E2 -13045.525} C_VEL
LIN {X 0,Y 360.263,Z 708.21,A -85,B 0,C 180,E1 -13047.764,E2 -13047.764} C_VEL
LIN {X 0,Y 360.241,Z 708.805,A -85,B 0,C 180,E1 -13050,E2 -13050} C_VEL
LIN {X 0,Y 360.265,Z 708.208,A -85,B 0,C 180,E1 -13052.236,E2 -13052.236} C_VEL
LIN {X 0,Y 360.323,Z 706.46,A -85,B 0,C 180,E1 -13054.475,E2 -13054.475} C_VEL
LIN {X 0,Y 360.483,Z 703.528,A -85,B 0,C 180,E1 -13056.718,E2 -13056.718} C_VEL
LIN {X 0,Y 360.78,Z 699.342,A -85,B 0,C 180,E1 -13058.966,E2 -13058.966} C_VEL
LIN {X 0,Y 361.273,Z 693.801,A -85,B 0,C 180,E1 -13061.218,E2 -13061.218} C_VEL
LIN {X 0,Y 362.147,Z 686.746,A -85,B 0,C 180,E1 -13063.467,E2 -13063.467} C_VEL
LIN {X 0,Y 363.188,Z 679.172,A -85,B 0,C 180,E1 -13065.431,E2 -13065.431} C_VEL
LIN {X 0,Y 364.537,Z 670.037,A -85,B 0,C 180,E1 -13067.387,E2 -13067.387} C_VEL
LIN {X 0,Y 365.986,Z 660.728,A -85,B 0,C 180,E1 -13069.054,E2 -13069.054} C_VEL
LIN {X 0,Y 367.714,Z 648.951,A -85,B 0,C 180,E1 -13070.809,E2 -13070.809} C_VEL
LIN {X 0,Y 369.55,Z 636.269,A -85,B 0,C 180,E1 -13072.356,E2 -13072.356} C_VEL
LIN {X 0,Y 371.153,Z 624.121,A -85,B 0,C 180,E1 -13073.579,E2 -13073.579} C_VEL
LIN {X 0,Y 372.902,Z 609.635,A -85,B 0,C 180,E1 -13074.751,E2 -13074.751} C_VEL
LIN {X 0,Y 374.17,Z 596.47,A -85,B 0,C 180,E1 -13075.595,E2 -13075.595} C_VEL
LIN {X 0,Y 376.529,Z 571.326,A -85,B 0,C 180,E1 -13076.838,E2 -13076.838} C_VEL
LIN {X 0,Y 377.936,Z 554.483,A -85,B 0,C 180,E1 -13077.441,E2 -13077.441} C_VEL
LIN {X 0,Y 383.088,Z 478.613,A -85,B 0,C 180,E1 -13079.616,E2 -13079.616} C_VEL
LIN {X 0,Y 386.61,Z 433.726,A -85,B 0,C 180,E1 -13080.993,E2 -13080.993} C_VEL
LIN {X 0,Y 385.334,Z 421.083,A -85,B 0,C 180,E1 -13081.77,E2 -13081.77} C_VEL
LIN {X 0,Y 384.103,Z 413.467,A -85,B 0,C 180,E1 -13082.343,E2 -13082.343} C_VEL
LIN {X 0,Y 380.772,Z 406.94,A -85,B 0,C 180,E1 -13083.299,E2 -13083.299} C_VEL
LIN {X 0,Y 378.572,Z 403.018,A -85,B 0,C 180,E1 -13083.964,E2 -13083.964} C_VEL
LIN {X 0,Y 376.474,Z 399.063,A -85,B 0,C 180,E1 -13084.708,E2 -13084.708} C_VEL
LIN {X 0,Y 375.095,Z 393.811,A -85,B 0,C 180,E1 -13086.839,E2 -13086.839} C_VEL
LIN {X 0,Y 373.919,Z 389.701,A -85,B 0,C 180,E1 -13088.989,E2 -13088.989} C_VEL
LIN {X 0,Y 372.81,Z 386.625,A -85,B 0,C 180,E1 -13091.285,E2 -13091.285} C_VEL
LIN {X 0,Y 372.354,Z 385.229,A -85,B 0,C 180,E1 -13092.804,E2 -13092.804} C_VEL
LIN {X 0,Y 372.009,Z 384.383,A -85,B 0,C 180,E1 -13094.348,E2 -13094.348} C_VEL
LIN {X 0,Y 371.818,Z 384.079,A -85,B 0,C 180,E1 -13095.912,E2 -13095.912} C_VEL
LIN {X 0,Y 371.863,Z 384.278,A -85,B 0,C 180,E1 -13097.483,E2 -13097.483} C_VEL
LIN {X 0,Y 372.322,Z 385.828,A -85,B 0,C 180,E1 -13100.075,E2 -13100.075} C_VEL
LIN {X 0,Y 373.081,Z 388.298,A -85,B 0,C 180,E1 -13102.297,E2 -13102.297} C_VEL
LIN {X 0,Y 373.975,Z 391.566,A -85,B 0,C 180,E1 -13104.368,E2 -13104.368} C_VEL
LIN {X 0,Y 375.027,Z 396.225,A -85,B 0,C 180,E1 -13106.619,E2 -13106.619} C_VEL
LIN {X 0,Y 375.741,Z 399.445,A -85,B 0,C 180,E1 -13107.851,E2 -13107.851} C_VEL
LIN {X 0,Y 379.283,Z 406.133,A -85,B 0,C 180,E1 -13109.086,E2 -13109.086} C_VEL
LIN {X 0,Y 382.205,Z 412.033,A -85,B 0,C 180,E1 -13109.998,E2 -13109.998} C_VEL
LIN {X 0,Y 384.697,Z 424.747,A -85,B 0,C 180,E1 -13111.109,E2 -13111.109} C_VEL
LIN {X 0,Y 386.245,Z 436.359,A -85,B 0,C 180,E1 -13111.93,E2 -13111.93} C_VEL
LIN {X 0,Y 379.473,Z 513.916,A -85,B 0,C 180,E1 -13114.458,E2 -13114.458} C_VEL
LIN {X 0,Y 376.926,Z 548.188,A -85,B 0,C 180,E1 -13115.599,E2 -13115.599} C_VEL
LIN {X 0,Y 375.456,Z 563.81,A -85,B 0,C 180,E1 -13116.35,E2 -13116.35} C_VEL
LIN {X 0,Y 373.773,Z 579.206,A -85,B 0,C 180,E1 -13117.354,E2 -13117.354} C_VEL
LIN {X 0,Y 371.94,Z 593.364,A -85,B 0,C 180,E1 -13118.525,E2 -13118.525} C_VEL
LIN {X 0,Y 370.107,Z 606.426,A -85,B 0,C 180,E1 -13119.869,E2 -13119.869} C_VEL
LIN {X 0,Y 368.381,Z 618.21,A -85,B 0,C 180,E1 -13121.364,E2 -13121.364} C_VEL
LIN {X 0,Y 366.739,Z 628.892,A -85,B 0,C 180,E1 -13123.008,E2 -13123.008} C_VEL
LIN {X 0,Y 365.229,Z 637.827,A -85,B 0,C 180,E1 -13124.658,E2 -13124.658} C_VEL
LIN {X 0,Y 363.829,Z 646.429,A -85,B 0,C 180,E1 -13126.597,E2 -13126.597} C_VEL
LIN {X 0,Y 362.869,Z 652.468,A -85,B 0,C 180,E1 -13128.266,E2 -13128.266} C_VEL
LIN {X 0,Y 362.22,Z 657.445,A -85,B 0,C 180,E1 -13129.943,E2 -13129.943} C_VEL
LIN {X 0,Y 361.42,Z 662.562,A -85,B 0,C 180,E1 -13132.177,E2 -13132.177} C_VEL
LIN {X 0,Y 361.188,Z 664.519,A -85,B 0,C 180,E1 -13133.296,E2 -13133.296} C_VEL
LIN {X 0,Y 360.747,Z 667.322,A -85,B 0,C 180,E1 -13135.531,E2 -13135.531} C_VEL
LIN {X 0,Y 360.751,Z 668.167,A -85,B 0,C 180,E1 -13136.65,E2 -13136.65} C_VEL
LIN {X 0,Y 360.523,Z 668.802,A -85,B 0,C 180,E1 -13138.883,E2 -13138.883} C_VEL
LIN {X 0,Y 360.492,Z 667.989,A -85,B 0,C 180,E1 -13141.117,E2 -13141.117} C_VEL
LIN {X 0,Y 360.496,Z 667.032,A -85,B 0,C 180,E1 -13142.235,E2 -13142.235} C_VEL
LIN {X 0,Y 360.567,Z 663.985,A -85,B 0,C 180,E1 -13144.472,E2 -13144.472} C_VEL
LIN {X 0,Y 360.82,Z 659.383,A -85,B 0,C 180,E1 -13146.711,E2 -13146.711} C_VEL
LIN {X 0,Y 361.015,Z 654.854,A -85,B 0,C 180,E1 -13148.396,E2 -13148.396} C_VEL
LIN {X 0,Y 361.536,Z 648.209,A -85,B 0,C 180,E1 -13150.359,E2 -13150.359} C_VEL
LIN {X 0,Y 362.181,Z 639.92,A -85,B 0,C 180,E1 -13152.325,E2 -13152.325} C_VEL
LIN {X 0,Y 362.993,Z 631.288,A -85,B 0,C 180,E1 -13154.006,E2 -13154.006} C_VEL
LIN {X 0,Y 363.842,Z 620.893,A -85,B 0,C 180,E1 -13155.69,E2 -13155.69} C_VEL
LIN {X 0,Y 364.898,Z 609.409,A -85,B 0,C 180,E1 -13157.225,E2 -13157.225} C_VEL
LIN {X 0,Y 366.033,Z 596.692,A -85,B 0,C 180,E1 -13158.615,E2 -13158.615} C_VEL
LIN {X 0,Y 367.082,Z 584.279,A -85,B 0,C 180,E1 -13159.721,E2 -13159.721} C_VEL
LIN {X 0,Y 368.08,Z 570.385,A -85,B 0,C 180,E1 -13160.714,E2 -13160.714} C_VEL
LIN {X 0,Y 368.936,Z 555.872,A -85,B 0,C 180,E1 -13161.512,E2 -13161.512} C_VEL
LIN {X 0,Y 369.709,Z 540.31,A -85,B 0,C 180,E1 -13162.125,E2 -13162.125} C_VEL
LIN {X 0,Y 373.477,Z 430.609,A -85,B 0,C 180,E1 -13164.954,E2 -13164.954} C_VEL
LIN {X 0,Y 368.213,Z 398.084,A -85,B 0,C 180,E1 -13166.191,E2 -13166.191} C_VEL
LIN {X 0,Y 368.869,Z 390.995,A -85,B 0,C 180,E1 -13167.518,E2 -13167.518} C_VEL
LIN {X 0,Y 367.718,Z 384.713,A -85,B 0,C 180,E1 -13168.854,E2 -13168.854} C_VEL
LIN {X 0,Y 364.183,Z 369.581,A -85,B 0,C 180,E1 -13172.238,E2 -13172.238} C_VEL
LIN {X 0,Y 361.918,Z 360.242,A -85,B 0,C 180,E1 -13174.442,E2 -13174.442} C_VEL
LIN {X 0,Y 361.857,Z 360.037,A -85,B 0,C 180,E1 -13177.221,E2 -13177.221} C_VEL
LIN {X 0,Y 361.811,Z 360.039,A -85,B 0,C 180,E1 -13180.75,E2 -13180.75} C_VEL
LIN {X 0,Y 361.812,Z 360.038,A -85,B 0,C 180,E1 -13184.369,E2 -13184.369} C_VEL
LIN {X 0,Y 361.822,Z 360.026,A -85,B 0,C 180,E1 -13187.571,E2 -13187.571} C_VEL
LIN {X 0,Y 361.845,Z 360.063,A -85,B 0,C 180,E1 -13191.572,E2 -13191.572} C_VEL
LIN {X 0,Y 361.906,Z 360.382,A -85,B 0,C 180,E1 -13191.845,E2 -13191.845} C_VEL
LIN {X 0,Y 366.22,Z 374.037,A -85,B 0,C 180,E1 -13194.692,E2 -13194.692} C_VEL
LIN {X 0,Y 370.035,Z 388.239,A -85,B 0,C 180,E1 -13197.426,E2 -13197.426} C_VEL
LIN {X 0,Y 372.106,Z 396.631,A -85,B 0,C 180,E1 -13198.897,E2 -13198.897} C_VEL
LIN {X 0,Y 373.591,Z 400.965,A -85,B 0,C 180,E1 -13199.142,E2 -13199.142} C_VEL
LIN {X 0,Y 378.497,Z 426.213,A -85,B 0,C 180,E1 -13200.126,E2 -13200.126} C_VEL
LIN {X 0,Y 380.146,Z 435.741,A -85,B 0,C 180,E1 -13200.471,E2 -13200.471} C_VEL
LIN {X 0,Y 377.195,Z 555.364,A -85,B 0,C 180,E1 -13202.764,E2 -13202.764} C_VEL
LIN {X 0,Y 376.548,Z 571.569,A -85,B 0,C 180,E1 -13203.163,E2 -13203.163} C_VEL
LIN {X 0,Y 375.474,Z 587.067,A -85,B 0,C 180,E1 -13203.759,E2 -13203.759} C_VEL
LIN {X 0,Y 374.188,Z 601.82,A -85,B 0,C 180,E1 -13204.555,E2 -13204.555} C_VEL
LIN {X 0,Y 372.748,Z 615.253,A -85,B 0,C 180,E1 -13205.493,E2 -13205.493} C_VEL
LIN {X 0,Y 370.973,Z 629.127,A -85,B 0,C 180,E1 -13206.704,E2 -13206.704} C_VEL
LIN {X 0,Y 369.215,Z 641.749,A -85,B 0,C 180,E1 -13208.064,E2 -13208.064} C_VEL
LIN {X 0,Y 367.473,Z 653.366,A -85,B 0,C 180,E1 -13209.576,E2 -13209.576} C_VEL
LIN {X 0,Y 365.882,Z 663.96,A -85,B 0,C 180,E1 -13211.232,E2 -13211.232} C_VEL
LIN {X 0,Y 364.27,Z 674.31,A -85,B 0,C 180,E1 -13213.178,E2 -13213.178} C_VEL
LIN {X 0,Y 362.965,Z 682.918,A -85,B 0,C 180,E1 -13215.134,E2 -13215.134} C_VEL
LIN {X 0,Y 362.057,Z 690.082,A -85,B 0,C 180,E1 -13217.101,E2 -13217.101} C_VEL
LIN {X 0,Y 361.183,Z 696.71,A -85,B 0,C 180,E1 -13219.347,E2 -13219.347} C_VEL
LIN {X 0,Y 361.088,Z 697.686,A -85,B 0,C 180,E1 -13219.738,E2 -13219.738} C_VEL
LIN {X 0,Y 360.238,Z 699.813,A -85,B 0,C 180,E1 -13220.603,E2 -13220.603} C_VEL
LIN {X 0,Y 357.097,Z 702.892,A -85,B 0,C 180,E1 -13222.021,E2 -13222.021} C_VEL
LIN {X 0,Y 354.497,Z 704.961,A -85,B 0,C 180,E1 -13223.188,E2 -13223.188} C_VEL
LIN {X 0,Y 353.359,Z 706.264,A -85,B 0,C 180,E1 -13224.108,E2 -13224.108} C_VEL
LIN {X 0,Y 353.251,Z 706.641,A -85,B 0,C 180,E1 -13224.422,E2 -13224.422} C_VEL
LIN {X 0,Y 353.184,Z 708.833,A -85,B 0,C 180,E1 -13226.577,E2 -13226.577} C_VEL
LIN {X 0,Y 353.145,Z 710.023,A -85,B 0,C 180,E1 -13228.86,E2 -13228.86} C_VEL
LIN {X 0,Y 353.145,Z 710.036,A -85,B 0,C 180,E1 -13231.14,E2 -13231.14} C_VEL
LIN {X 0,Y 353.186,Z 708.899,A -85,B 0,C 180,E1 -13233.422,E2 -13233.422} C_VEL
LIN {X 0,Y 353.314,Z 706.29,A -85,B 0,C 180,E1 -13235.965,E2 -13235.965} C_VEL
LIN {X 0,Y 353.643,Z 702.075,A -85,B 0,C 180,E1 -13238.572,E2 -13238.572} C_VEL
LIN {X 0,Y 354.121,Z 696.945,A -85,B 0,C 180,E1 -13240.867,E2 -13240.867} C_VEL
LIN {X 0,Y 355.043,Z 690.376,A -85,B 0,C 180,E1 -13243.158,E2 -13243.158} C_VEL
LIN {X 0,Y 356.014,Z 683.284,A -85,B 0,C 180,E1 -13245.163,E2 -13245.163} C_VEL
LIN {X 0,Y 357.36,Z 674.76,A -85,B 0,C 180,E1 -13247.157,E2 -13247.157} C_VEL
LIN {X 0,Y 358.766,Z 666.103,A -85,B 0,C 180,E1 -13248.858,E2 -13248.858} C_VEL
LIN {X 0,Y 360.465,Z 655.34,A -85,B 0,C 180,E1 -13250.632,E2 -13250.632} C_VEL
LIN {X 0,Y 362.33,Z 643.684,A -85,B 0,C 180,E1 -13252.224,E2 -13252.224} C_VEL
LIN {X 0,Y 364.164,Z 631.462,A -85,B 0,C 180,E1 -13253.606,E2 -13253.606} C_VEL
LIN {X 0,Y 365.963,Z 618.117,A -85,B 0,C 180,E1 -13254.84,E2 -13254.84} C_VEL
LIN {X 0,Y 367.626,Z 603.628,A -85,B 0,C 180,E1 -13255.908,E2 -13255.908} C_VEL
LIN {X 0,Y 368.927,Z 589.033,A -85,B 0,C 180,E1 -13256.743,E2 -13256.743} C_VEL
LIN {X 0,Y 370.084,Z 574.422,A -85,B 0,C 180,E1 -13257.344,E2 -13257.344} C_VEL
LIN {X 0,Y 370.884,Z 558.274,A -85,B 0,C 180,E1 -13257.777,E2 -13257.777} C_VEL
LIN {X 0,Y 373.99,Z 436.562,A -85,B 0,C 180,E1 -13260.149,E2 -13260.149} C_VEL
LIN {X 0,Y 369.181,Z 410.41,A -85,B 0,C 180,E1 -13261.162,E2 -13261.162} C_VEL
LIN {X 0,Y 367.201,Z 401.705,A -85,B 0,C 180,E1 -13261.544,E2 -13261.544} C_VEL
LIN {X 0,Y 364.867,Z 396.225,A -85,B 0,C 180,E1 -13261.929,E2 -13261.929} C_VEL
LIN {X 0,Y 361.679,Z 383.494,A -85,B 0,C 180,E1 -13264.299,E2 -13264.299} C_VEL
LIN {X 0,Y 357.992,Z 370.766,A -85,B 0,C 180,E1 -13266.871,E2 -13266.871} C_VEL
LIN {X 0,Y 354.819,Z 361.072,A -85,B 0,C 180,E1 -13269.01,E2 -13269.01} C_VEL
LIN {X 0,Y 354.785,Z 360.912,A -85,B 0,C 180,E1 -13272.866,E2 -13272.866} C_VEL
LIN {X 0,Y 354.765,Z 360.922,A -85,B 0,C 180,E1 -13276.103,E2 -13276.103} C_VEL
LIN {X 0,Y 354.765,Z 360.922,A -85,B 0,C 180,E1 -13279.176,E2 -13279.176} C_VEL
LIN {X 0,Y 354.798,Z 360.917,A -85,B 0,C 180,E1 -13282.404,E2 -13282.404} C_VEL
LIN {X 0,Y 354.808,Z 360.904,A -85,B 0,C 180,E1 -13284.94,E2 -13284.94} C_VEL
LIN {X 0,Y 354.793,Z 360.903,A -85,B 0,C 180,E1 -13288.405,E2 -13288.405} C_VEL
LIN {X 0,Y 354.801,Z 360.908,A -85,B 0,C 180,E1 -13291.615,E2 -13291.615} C_VEL
LIN {X 0,Y 354.841,Z 360.911,A -85,B 0,C 180,E1 -13295.422,E2 -13295.422} C_VEL
LIN {X 0,Y 354.827,Z 360.902,A -85,B 0,C 180,E1 -13299.113,E2 -13299.113} C_VEL
LIN {X 0,Y 354.88,Z 360.888,A -85,B 0,C 180,E1 -13302.719,E2 -13302.719} C_VEL
LIN {X 0,Y 354.952,Z 360.895,A -85,B 0,C 180,E1 -13306.255,E2 -13306.255} C_VEL
LIN {X 0,Y 354.956,Z 360.878,A -85,B 0,C 180,E1 -13309.735,E2 -13309.735} C_VEL
LIN {X 0,Y 355.113,Z 360.872,A -85,B 0,C 180,E1 -13313.18,E2 -13313.18} C_VEL
LIN {X 0,Y 355.234,Z 360.862,A -85,B 0,C 180,E1 -13317.732,E2 -13317.732} C_VEL
LIN {X 0,Y 355.374,Z 360.833,A -85,B 0,C 180,E1 -13320,E2 -13320} C_VEL
LIN {X 0,Y 355.242,Z 360.842,A -85,B 0,C 180,E1 -13322.268,E2 -13322.268} C_VEL
LIN {X 0,Y 355.1,Z 360.861,A -85,B 0,C 180,E1 -13326.82,E2 -13326.82} C_VEL
LIN {X 0,Y 354.957,Z 360.891,A -85,B 0,C 180,E1 -13330.265,E2 -13330.265} C_VEL
LIN {X 0,Y 354.943,Z 360.875,A -85,B 0,C 180,E1 -13334.019,E2 -13334.019} C_VEL
LIN {X 0,Y 354.89,Z 360.896,A -85,B 0,C 180,E1 -13338.092,E2 -13338.092} C_VEL
LIN {X 0,Y 354.836,Z 360.909,A -85,B 0,C 180,E1 -13342.106,E2 -13342.106} C_VEL
LIN {X 0,Y 354.899,Z 360.892,A -85,B 0,C 180,E1 -13345.827,E2 -13345.827} C_VEL
LIN {X 0,Y 354.854,Z 360.893,A -85,B 0,C 180,E1 -13349.678,E2 -13349.678} C_VEL
LIN {X 0,Y 354.806,Z 360.905,A -85,B 0,C 180,E1 -13353.702,E2 -13353.702} C_VEL
LIN {X 0,Y 354.797,Z 360.915,A -85,B 0,C 180,E1 -13356.459,E2 -13356.459} C_VEL
LIN {X 0,Y 354.824,Z 360.87,A -85,B 0,C 180,E1 -13359.424,E2 -13359.424} C_VEL
LIN {X 0,Y 354.788,Z 360.911,A -85,B 0,C 180,E1 -13362.867,E2 -13362.867} C_VEL
LIN {X 0,Y 354.766,Z 360.887,A -85,B 0,C 180,E1 -13366.104,E2 -13366.104} C_VEL
LIN {X 0,Y 354.788,Z 360.916,A -85,B 0,C 180,E1 -13369.179,E2 -13369.179} C_VEL
LIN {X 0,Y 354.852,Z 361.081,A -85,B 0,C 180,E1 -13372.572,E2 -13372.572} C_VEL
LIN {X 0,Y 359.019,Z 376.612,A -85,B 0,C 180,E1 -13375.894,E2 -13375.894} C_VEL
LIN {X 0,Y 361.11,Z 384.629,A -85,B 0,C 180,E1 -13377.475,E2 -13377.475} C_VEL
LIN {X 0,Y 363.775,Z 391.883,A -85,B 0,C 180,E1 -13378.218,E2 -13378.218} C_VEL
LIN {X 0,Y 368.349,Z 402.278,A -85,B 0,C 180,E1 -13378.893,E2 -13378.893} C_VEL
LIN {X 0,Y 373.404,Z 433.68,A -85,B 0,C 180,E1 -13380.046,E2 -13380.046} C_VEL
LIN {X 0,Y 370.029,Z 564.717,A -85,B 0,C 180,E1 -13382.614,E2 -13382.614} C_VEL
LIN {X 0,Y 369.11,Z 580.117,A -85,B 0,C 180,E1 -13383.115,E2 -13383.115} C_VEL
LIN {X 0,Y 367.809,Z 595.575,A -85,B 0,C 180,E1 -13383.853,E2 -13383.853} C_VEL
LIN {X 0,Y 366.426,Z 610.202,A -85,B 0,C 180,E1 -13384.811,E2 -13384.811} C_VEL
LIN {X 0,Y 364.598,Z 624.28,A -85,B 0,C 180,E1 -13385.971,E2 -13385.971} C_VEL
LIN {X 0,Y 362.753,Z 637.638,A -85,B 0,C 180,E1 -13387.353,E2 -13387.353} C_VEL
LIN {X 0,Y 360.923,Z 649.766,A -85,B 0,C 180,E1 -13388.885,E2 -13388.885} C_VEL
LIN {X 0,Y 359.241,Z 660.818,A -85,B 0,C 180,E1 -13390.575,E2 -13390.575} C_VEL
LIN {X 0,Y 357.716,Z 670.119,A -85,B 0,C 180,E1 -13392.27,E2 -13392.27} C_VEL
LIN {X 0,Y 356.249,Z 679.237,A -85,B 0,C 180,E1 -13394.261,E2 -13394.261} C_VEL
LIN {X 0,Y 355.194,Z 686.797,A -85,B 0,C 180,E1 -13396.265,E2 -13396.265} C_VEL
LIN {X 0,Y 354.266,Z 693.849,A -85,B 0,C 180,E1 -13398.558,E2 -13398.558} C_VEL
LIN {X 0,Y 353.741,Z 699.385,A -85,B 0,C 180,E1 -13400.855,E2 -13400.855} C_VEL
LIN {X 0,Y 353.395,Z 703.558,A -85,B 0,C 180,E1 -13403.147,E2 -13403.147} C_VEL
LIN {X 0,Y 353.238,Z 706.48,A -85,B 0,C 180,E1 -13405.436,E2 -13405.436} C_VEL
LIN {X 0,Y 353.171,Z 708.224,A -85,B 0,C 180,E1 -13407.719,E2 -13407.719} C_VEL
LIN {X 0,Y 353.141,Z 708.818,A -85,B 0,C 180,E1 -13410,E2 -13410} C_VEL
LIN {X 0,Y 353.173,Z 708.221,A -85,B 0,C 180,E1 -13412.281,E2 -13412.281} C_VEL
LIN {X 0,Y 353.238,Z 706.474,A -85,B 0,C 180,E1 -13414.565,E2 -13414.565} C_VEL
LIN {X 0,Y 353.396,Z 703.542,A -85,B 0,C 180,E1 -13416.853,E2 -13416.853} C_VEL
LIN {X 0,Y 353.741,Z 699.356,A -85,B 0,C 180,E1 -13419.146,E2 -13419.146} C_VEL
LIN {X 0,Y 354.271,Z 693.815,A -85,B 0,C 180,E1 -13421.442,E2 -13421.442} C_VEL
LIN {X 0,Y 355.193,Z 686.761,A -85,B 0,C 180,E1 -13423.736,E2 -13423.736} C_VEL
LIN {X 0,Y 356.476,Z 677.962,A -85,B 0,C 180,E1 -13426.023,E2 -13426.023} C_VEL
LIN {X 0,Y 357.91,Z 668.575,A -85,B 0,C 180,E1 -13428.015,E2 -13428.015} C_VEL
LIN {X 0,Y 359.701,Z 657.629,A -85,B 0,C 180,E1 -13429.926,E2 -13429.926} C_VEL
LIN {X 0,Y 361.379,Z 646.634,A -85,B 0,C 180,E1 -13431.521,E2 -13431.521} C_VEL
LIN {X 0,Y 363.176,Z 635.009,A -85,B 0,C 180,E1 -13432.92,E2 -13432.92} C_VEL
LIN {X 0,Y 364.857,Z 622.602,A -85,B 0,C 180,E1 -13434.163,E2 -13434.163} C_VEL
LIN {X 0,Y 366.432,Z 609.843,A -85,B 0,C 180,E1 -13435.204,E2 -13435.204} C_VEL
LIN {X 0,Y 367.824,Z 596.042,A -85,B 0,C 180,E1 -13436.1,E2 -13436.1} C_VEL
LIN {X 0,Y 369.765,Z 579.969,A -85,B 0,C 180,E1 -13437.063,E2 -13437.063} C_VEL
LIN {X 0,Y 371.523,Z 563.273,A -85,B 0,C 180,E1 -13437.802,E2 -13437.802} C_VEL
LIN {X 0,Y 373.596,Z 536.036,A -85,B 0,C 180,E1 -13438.628,E2 -13438.628} C_VEL
LIN {X 0,Y 378.831,Z 467.988,A -85,B 0,C 180,E1 -13440.677,E2 -13440.677} C_VEL
LIN {X 0,Y 381.652,Z 435.276,A -85,B 0,C 180,E1 -13441.717,E2 -13441.717} C_VEL
LIN {X 0,Y 380.539,Z 422.876,A -85,B 0,C 180,E1 -13442.517,E2 -13442.517} C_VEL
LIN {X 0,Y 379.664,Z 417.463,A -85,B 0,C 180,E1 -13442.959,E2 -13442.959} C_VEL
LIN {X 0,Y 375.965,Z 409.877,A -85,B 0,C 180,E1 -13444.125,E2 -13444.125} C_VEL
LIN {X 0,Y 372.307,Z 403.685,A -85,B 0,C 180,E1 -13445.358,E2 -13445.358} C_VEL
LIN {X 0,Y 369.728,Z 399.126,A -85,B 0,C 180,E1 -13446.443,E2 -13446.443} C_VEL
LIN {X 0,Y 368.555,Z 394.869,A -85,B 0,C 180,E1 -13448.572,E2 -13448.572} C_VEL
LIN {X 0,Y 367.605,Z 391.991,A -85,B 0,C 180,E1 -13450.544,E2 -13450.544} C_VEL
LIN {X 0,Y 366.743,Z 389.466,A -85,B 0,C 180,E1 -13453.264,E2 -13453.264} C_VEL
LIN {X 0,Y 366.39,Z 388.699,A -85,B 0,C 180,E1 -13455.213,E2 -13455.213} C_VEL
LIN {X 0,Y 366.407,Z 388.93,A -85,B 0,C 180,E1 -13457.83,E2 -13457.83} C_VEL
LIN {X 0,Y 366.774,Z 390.252,A -85,B 0,C 180,E1 -13460.038,E2 -13460.038} C_VEL
LIN {X 0,Y 367.469,Z 392.631,A -85,B 0,C 180,E1 -13462.265,E2 -13462.265} C_VEL
LIN {X 0,Y 368.313,Z 396.034,A -85,B 0,C 180,E1 -13464.454,E2 -13464.454} C_VEL
LIN {X 0,Y 369.161,Z 399.58,A -85,B 0,C 180,E1 -13466.141,E2 -13466.141} C_VEL
LIN {X 0,Y 372.899,Z 406.249,A -85,B 0,C 180,E1 -13467.662,E2 -13467.662} C_VEL
LIN {X 0,Y 375.792,Z 411.781,A -85,B 0,C 180,E1 -13468.69,E2 -13468.69} C_VEL
LIN {X 0,Y 378.074,Z 416.706,A -85,B 0,C 180,E1 -13469.464,E2 -13469.464} C_VEL
LIN {X 0,Y 380.337,Z 429.889,A -85,B 0,C 180,E1 -13470.623,E2 -13470.623} C_VEL
LIN {X 0,Y 381.279,Z 437.632,A -85,B 0,C 180,E1 -13471.193,E2 -13471.193} C_VEL
LIN {X 0,Y 373.764,Z 517.764,A -85,B 0,C 180,E1 -13473.889,E2 -13473.889} C_VEL
LIN {X 0,Y 371.276,Z 548.36,A -85,B 0,C 180,E1 -13474.942,E2 -13474.942} C_VEL
LIN {X 0,Y 369.665,Z 564.304,A -85,B 0,C 180,E1 -13475.725,E2 -13475.725} C_VEL
LIN {X 0,Y 368.019,Z 578.547,A -85,B 0,C 180,E1 -13476.669,E2 -13476.669} C_VEL
LIN {X 0,Y 366.01,Z 592.899,A -85,B 0,C 180,E1 -13477.863,E2 -13477.863} C_VEL
LIN {X 0,Y 364.011,Z 606.054,A -85,B 0,C 180,E1 -13479.221,E2 -13479.221} C_VEL
LIN {X 0,Y 362.175,Z 617.938,A -85,B 0,C 180,E1 -13480.738,E2 -13480.738} C_VEL
LIN {X 0,Y 360.367,Z 628.69,A -85,B 0,C 180,E1 -13482.405,E2 -13482.405} C_VEL
LIN {X 0,Y 358.7,Z 637.707,A -85,B 0,C 180,E1 -13484.08,E2 -13484.08} C_VEL
LIN {X 0,Y 357.189,Z 646.375,A -85,B 0,C 180,E1 -13486.053,E2 -13486.053} C_VEL
LIN {X 0,Y 355.977,Z 653.398,A -85,B 0,C 180,E1 -13488.036,E2 -13488.036} C_VEL
LIN {X 0,Y 355.283,Z 658.25,A -85,B 0,C 180,E1 -13489.745,E2 -13489.745} C_VEL
LIN {X 0,Y 354.434,Z 663.256,A -85,B 0,C 180,E1 -13492.022,E2 -13492.022} C_VEL
LIN {X 0,Y 354.177,Z 665.16,A -85,B 0,C 180,E1 -13493.162,E2 -13493.162} C_VEL
